// TwinCAT 3 PLC project Area2
// ProgramVersion: 3.1.4023.0
// libraries:
//   Tc2_DataExchange, * (Beckhoff Automation GmbH)
//   Tc2_MC2, * (Beckhoff Automation GmbH)
//   Tc2_Standard, * (Beckhoff Automation GmbH)
//   Tc2_System, * (Beckhoff Automation GmbH)
//   Tc2_TcpIp, * (Beckhoff Automation GmbH)
//   Tc2_Utilities, * (Beckhoff Automation GmbH)
//   Tc3_BA_Common, * (Beckhoff Automation GmbH)
//   Tc3_Database, * (Beckhoff Automation GmbH)
//   Tc3_JsonXml, * (Beckhoff Automation GmbH)
//   Tc3_Module, * (Beckhoff Automation GmbH)
//   Tc3_PackML_V2, * (Beckhoff Automation GmbH)
// project tree:
//   COMMs_ADS/ AdsClient.TcPOU (not stored), AdsHandle.TcPOU
//   COMMs_ADS/PROTOTYPE/ AdsClient_1.TcPOU (not stored), AdsHandle_1.TcPOU (not stored)
//   COMMs_TCP/ TcpServer1Vision.TcPOU
//   COMMs_TCP/Types/ DUT.TcDUT, TcpData.TcDUT (not stored), TcpDataQueue.TcPOU
//   DUTs/Enums/ E_PMLCustomUnitMode.TcDUT (not stored), InsertionDirection.TcDUT, SectionEnum.TcDUT (not stored), SectionTask.TcDUT (not stored), ConveyorMode.TcDUT (not stored), Cover.TcDUT (not stored), EventsEnum.TcTLEO (not stored), MaterialEnums.TcDUT, MaterialType.TcDUT (not stored), Surface.TcDUT (not stored)
//   DUTs/Enums/Materials/ Cardboard.TcDUT, Chipboard.TcDUT, CornerGuard.TcDUT (not stored), WoodBunk.TcDUT (not stored)
//   DUTs/Enums/Robot Tasks/ TaskA22.TcDUT (not stored), TaskA26.TcDUT, TaskA21.TcDUT
//   DUTs/Hardware/ A21ToolStorage.TcDUT (not stored), ConveyorLSC.TcPOU (not stored), ConveyorSC.TcPOU (not stored), FoldingMachine.TcDUT (not stored), PMLStackLight.TcPOU (not stored), Conveyor.TcPOU (not stored)
//   DUTs/Hardware/Big Machines/ StrapMachine.TcPOU (not stored), WrapMachine.TcPOU
//   DUTs/Hardware/Insertion Package/Drives/ AirPiston.TcPOU (not stored), ClearLinkMC.TcPOU, ServoNC.TcPOU (not stored), SimplePiston.TcPOU (not stored)
//   DUTs/Hardware/Insertion Package/ Homing.TcDUT (not stored), Insertion.TcPOU, SuctionPad.TcDUT (not stored)
//   DUTs/Hardware/Insertion Package/Prototypes/ FBA_Drive.TcPOU (not stored), FBA_TrifectaDrive.TcPOU (not stored), I_ContinuousDrive.TcIO (not stored), I_Drive.TcIO (not stored), I_EncodedDrive.TcIO, I_PositionalDrive.TcIO (not stored)
//   DUTs/Hardware/Material Holders/ MaterialHolder.TcPOU (not stored), MaterialSlot.TcDUT (not stored), SkidMagazine.TcPOU (not stored), StagingTable.TcPOU
//   DUTs/Hardware/Robots/ KukaRobot.TcPOU, RobotA21.TcPOU (not stored), RobotA26.TcPOU, RobotA22.TcPOU (not stored)
//   DUTs/ Watchdog.TcPOU, ONE_BIT.TcDUT (not stored), VisionFrame.TcDUT (not stored), VisionSuite.TcDUT (not stored)
//   COMMs_ADS/Types/ AdsSocket.TcPOU (not stored), AdsDataQueue.TcPOU, AdsData.TcDUT
//   DUTs/Bundle/ Bundle.TcDUT, CardboardMaterial.TcDUT, Interval.TcDUT, Material.TcDUT, PositionMaterials.TcDUT (not stored)
//   DUTs/Containers/ DynamicQueue.TcPOU, PtrQueue.TcPOU, IntQueue.TcPOU, Queue.TcPOU, StringQueue.TcPOU
//   EventLogging/ EventLogger.TcIO, SqlDatabaseAccessor.TcPOU (not stored)
//   / GlobalTextList.TcGTLO (not stored), PlcTask.TcTTO (not stored)
//   GVLs/ GVL.TcGVL, CONSTS.TcGVL
//   HARDWARE_DISTRUBUTION/ ConveyorControlModule.TcPOU, ConveyorSyncUnit.TcPOU, A21.TcPOU, A22.TcPOU, A23.TcPOU, A24.TcPOU, A25.TcPOU, A26.TcPOU
//   POUs/Helper Functions/Document/ CreateJsonDocumentManual.TcPOU (not stored), CreateJsonDocumentAuto.TcPOU (not stored), FrameIsValid.TcPOU (not stored), VisionJsonParser.TcPOU (not stored)
//   POUs/Helper Functions/General/ BufferIsEmpty.TcPOU, BundleIsValid.TcPOU (not stored), InRange.TcPOU (not stored), PositionIsValid.TcPOU (not stored), TimestructToString.TcPOU
//   POUs/Helper Functions/Hardware Modules/ InsertionQuality.TcPOU (not stored), SetSuctions.TcPOU, SetSuctionsPtr.TcPOU, SetupHardware.TcPOU, SuctionQuality.TcPOU (not stored), SuctionQualityPtr.TcPOU
//   POUs/Helper Functions/Material Functions/ GetPairMasterLength.TcPOU, GetMaterialLength.TcPOU, MatchesMaterialType.TcPOU (not stored)
//   POUs/Helper Functions/Other/ ForceSetLifterConveyors.TcPOU (not stored), SizeCheck.TcPOU (not stored)
//   POUs/Helper Functions/Utility/ AddToStringArray.TcPOU (not stored), DataIsEmpty.TcPOU (not stored), CleanStringsArray.TcPOU (not stored), IntegerBitAccess.TcPOU (not stored), IntegerToBoolArray.TcPOU (not stored), JoinStrings.TcPOU (not stored), WithinTolerance.TcPOU (not stored)
//   POUs/ MAIN.TcPOU
//   Sections/A21a - Chipboard/AOIs/ AOI_LoadChipboard.TcPOU
//   Sections/A21a - Chipboard/ ChipboardEx.TcPOU
//   Sections/A21b - Wood Bunk/AOIs/ AOI_LoadWoodBunk.TcPOU, AOI_StageWoodBunk.TcPOU (not stored), AOI_StagingTemplate.TcPOU
//   Sections/A21b - Wood Bunk/ WoodBunkEx.TcPOU
//   Sections/A22 - Cardboard/AOIs/ AOI_LoadCornerCardboard.TcPOU, AOI_LoadCornerGuard.TcPOU, AOI_LoadFlatCardboard.TcPOU
//   Sections/A22 - Cardboard/ CardboardEx.TcPOU
//   Sections/A26 - Spacer Recollection/ SpacerRecollectionUnit.TcPOU
//   Sections/Abstract/ SectionEx.TcPOU
// real-time tasks:
//   TASK PlcTask: cycle T#10ms, priority 20, ADS port 350

// ---- COMMs_TCP/Types/DUT.TcDUT
TYPE DUT :
UNION
END_UNION
END_TYPE

// ---- DUTs/Enums/InsertionDirection.TcDUT
{attribute 'qualified_only'}
{attribute 'strict'}
TYPE InsertionDirection :
(
	IN,
	OUT,
	
	size
);
END_TYPE

// ---- DUTs/Enums/Materials/Cardboard.TcDUT
{attribute 'qualified_only'}
{attribute 'to_string'}
TYPE Cardboard :
(
	CAR20S := 1,
	CAR20M,
	CAR20L,
	
	CAR28S,
	CAR28M,
	CAR28L,
	
	size
);
END_TYPE

// ---- DUTs/Enums/Materials/Chipboard.TcDUT
{attribute 'qualified_only'}
{attribute 'to_string'}
TYPE Chipboard :
(
	CIP18 := 1,
	CIP54,
	
	size
);
END_TYPE

// ---- DUTs/Enums/Robot Tasks/TaskA26.TcDUT
{attribute 'qualified_only'}
{attribute 'to_string'}
//{attribute 'strict'}
TYPE TaskA26 :
(
	IDLE,
	PICK_SPACER,
	
	size
);
END_TYPE

// ---- DUTs/Enums/Robot Tasks/TaskA21.TcDUT
{attribute 'qualified_only'}
//{attribute 'strict'}
{attribute 'to_string'}
TYPE TaskA21 :
(
	IDLE,
	STAGE_BUNK,
	REMOVE_BUNK_FROM_STAGE,
	
	LOAD_BUNK_TOP := 4,
	LOAD_BUNK_SIDE,
	LOAD_BUNK_BOTTOM,
	REMOVE_BUNK_TOP,
	REMOVE_BUNK_SIDE,
	REMOVE_BUNK_BOTTOM,
	
	//GET_CHIPBOARD_FROM_SKID := 11,
	//OFFLOAD_CHIPBOARD,
	PLACE_CHIPBOARD_TOP := 13,
	PLACE_CHIPBOARD_BOTTOM,
	REMOVE_CHIPBOARD_TOP,
	REMOVE_CHIPBOARD_BOTTOM,
	
	FIX_CHIPBOARD_ORIENTATION := 19,
	
	//testing only
	MOVE_HOME := 21,
	MOVE_POSITION1,
	MOVE_POSITION2,
	MOVE_UP,
	MOVE_DOWN,
	
	DIRECT_BUNK_TOP := 27,
	DIRECT_BUNK_SIDE,
	DIRECT_BUNK_BOTTOM,
	
	INSPECT_BUNK := 31,
	INSPECT_CHIPBOARD,
	
	TOOL_CHANGE_BUNK := 34,
	TOOL_CHANGE_CHIPBOARD,
	
	size
);
END_TYPE

// ---- COMMs_ADS/Types/AdsData.TcDUT
{attribute 'enable_dynamic_creation'}
TYPE AdsData :
STRUCT	
	description : EventsEnum; //purpose
	
	timestamp : TIMESTRUCT; //relevant timestamp (ex: arrival time)
	
	binaryData : ARRAY[0..100000] OF BYTE; //contents
END_STRUCT
END_TYPE

// ---- DUTs/Bundle/Bundle.TcDUT
{attribute 'enable_dynamic_creation'}
TYPE Bundle :
STRUCT
	id : STRING;
	weight : REAL;
	
	length : INT;
	width : INT;
	height : INT;
	
	pieces : INT;
	layers : INT;
	piecesPerLayer : INT;
	
	extrusionWeight : INT;
	extrusionHeight : INT;
	extrusionWidth : INT;
	
	//if a process is true, send it to the correct area and turn it false when complete
	reqProcesses : ARRAY[0..3] OF BOOL;
	
	manRE, autoRE : BOOL; //repacking - coming soon
	manSS, autoSS : BOOL; //packaging
	
	currStep : USINT; //for runtime use only
	
	paperFront : BOOL;
	paperBack : BOOL;
	cardboardFront : BOOL;
	cardboardBack : BOOL;
	
	paperTop : ARRAY[0..Consts.maxPairs] OF Interval;
	paperLeft : ARRAY[0..Consts.maxPairs] OF Interval;
	paperRight : ARRAY[0..Consts.maxPairs] OF Interval;
	paperBottom : ARRAY[0..Consts.maxPairs] OF Interval;
		
	cardboard : ARRAY[0..Consts.maxPairs] OF PositionMaterials;
	cardboardFolds : ARRAY[Surface.TOP_LEFT..Surface.BOTTOM_RIGHT] OF ARRAY[0..Consts.maxPairs] OF INT;
	
	topLeftFolds : ARRAY[0..Consts.maxPairs] OF INT;
	topRightFolds : ARRAY[0..Consts.maxPairs] OF INT;
	bottomLeftFolds : ARRAY[0..Consts.maxPairs] OF INT;
	bottomRightFolds : ARRAY[0..Consts.maxPairs] OF INT;
	
	cornerGuard : ARRAY[0..Consts.maxPairs] OF PositionMaterials;
	
	chipboard : ARRAY[0..Consts.maxPairs] OF PositionMaterials;
	woodBunk : ARRAY[0..Consts.maxPairs] OF PositionMaterials;
	
	cardboard_over_cornerGuard : BOOL;
	
	//for production log database
	timeStart : TIMESTRUCT;
	timeDone : TIMESTRUCT;
END_STRUCT
END_TYPE

// ---- DUTs/Bundle/CardboardMaterial.TcDUT
TYPE CardboardMaterial :
STRUCT
	foldType : (FLAT, CORNER, COVER);
	foldPos1 : REAL;
	foldPos2 : REAL;
END_STRUCT
END_TYPE

// ---- DUTs/Bundle/Interval.TcDUT
TYPE Interval :
STRUCT
	startPos : INT;
	endPos : INT;
END_STRUCT
END_TYPE

// ---- DUTs/Bundle/Material.TcDUT
TYPE Material :
STRUCT
	code : STRING;
	width : REAL;
	length : REAL;
END_STRUCT
END_TYPE
(*
use this struct to keep track of where materials are
materials enter the system when pulled from their magazine/skid and exit the system when placed on the bundle or otherwise lost
*)

// ---- DUTs/Enums/MaterialEnums.TcDUT
{attribute 'qualified_only'}
{attribute 'strict'}
{attribute 'to_string'}
TYPE MaterialEnums :
(
	//CARDBOARD - 6 x 3
	CAR20S, CAR20M, CAR20L, CAR28S, CAR28M, CAR28L, //base (flat)
	CAR20SF, CAR20MF, CAR20LF, CAR28SF, CAR28MF, CAR28LF, //single folded (L shape) - F
	CAR20SD, CAR20MD, CAR20LD, CAR28SD, CAR28MD, CAR28LD, //double folded (C shape) - D
	
	//CHIPBOARD - 2
	CIP18, CIP54,
	
	//CORNER BOARD - 2
	COR48, COR96,
	
	//PAPER - 1
	PAP28,
	
	//WOOD BUNK - 21
	WDT20, WDT22, WDT28, //top
	WDB20, WDB22, WDB28, //bottom
	WDS08, WDS10, WDS12, WDS14, WDS20, WDS22, WDS28, //side
	WDS8X8, WDS8X10, WDS12X12, WDS12X14, WDS20X10, WDS20X12, //side combined - X
	WDW20, WDW22, //special top (wide)
	
	size //number of materials
);
END_TYPE

// ---- GVLs/GVL.TcGVL
{attribute 'qualified_only'}
VAR_GLOBAL
	bundleOut : Bundle; //may or may not be used?
	
	iecCriticalSection : FB_IecCriticalSection; //must be used if communication routines are separated into their own core/task
END_VAR

// ---- GVLs/CONSTS.TcGVL
{attribute 'qualified_only'}
VAR_GLOBAL CONSTANT
	maxPairs : USINT := 16;
	initArraySize : USINT := 4;
	maxQueue : INT := 16;
	
	nullPos : REAL := -1;
	
	numMaterials : INT := 32;
	allMaterials : ARRAY[0..numMaterials] OF Material := [
		(code := '', width := 0, length := 0), //null material
		(code := 'PAP28', width := 28, length := -1),
		
		(code := 'CAR20S', width := 20, length := 30),
		(code := 'CAR20M', width := 20, length := 45),
		(code := 'CAR20L', width := 20, length := 60),
		(code := 'CAR28S', width := 28, length := 30),
		(code := 'CAR28M', width := 28, length := 45),
		(code := 'CAR28L', width := 28, length := 60),
		
		(code := 'COR48', width := 1.5, length := 48),
		(code := 'COR96', width := 1.5, length := 96),
		
		(code := 'CIP18', width := 20, length := 18),
		(code := 'CIP54', width := 20, length := 54),
		
		(code := 'WDT20', width := 20, length := 2.5),
		(code := 'WDT22', width := 22, length := 2.5),
		(code := 'WDT28', width := 28, length := 2.5),
		
		(code := 'WDB20', width := 20, length := 2.5),
		(code := 'WDB22', width := 22, length := 2.5),
		(code := 'WDB28', width := 28, length := 2.5),
		
		(code := 'WDS08', width := 8, length := 2.5),
		(code := 'WDS10', width := 10, length := 2.5),
		(code := 'WDS12', width := 12, length := 2.5),
		(code := 'WDS14', width := 14, length := 2.5),
		(code := 'WDS8x8', width := 16, length := 2.5),
		(code := 'WDS8x10', width := 18, length := 2.5),
		(code := 'WDS20', width := 20, length := 2.5),
		(code := 'WDS22', width := 22, length := 2.5),
		(code := 'WDS12x12', width := 24, length := 2.5),
		(code := 'WDS12x14', width := 26, length := 2.5),
		(code := 'WDS28', width := 28, length := 2.5),
		(code := 'WDS20x10', width := 30, length := 2.5),
		(code := 'WDS20x12', width := 32, length := 2.5),
		
		(code := 'WDW20', width := 20, length := 6),
		(code := 'WDW22', width := 22, length := 6)];

	//nullBundle : Bundle;
	
	//conveyorLength : REAL := 0;
	precisionTolerance : REAL := 0.05 * 25.4;
END_VAR
VAR_GLOBAL CONSTANT
	numTotalConveyors : INT := 38;
	
	numCellConveyors : INT := 20;
	
	numReceiverConveyors : INT := 6;
	numOutputConveyors : INT := 12;
END_VAR

// ---- DUTs/Hardware/Insertion Package/Prototypes/I_EncodedDrive.TcIO
INTERFACE I_EncodedDrive EXTENDS I_PositionalDrive, I_ContinuousDrive
//this drive can perform absolute/relative targeting and continuous motion
//only used if a drive with both encoded and continuous behavior is needed

END_INTERFACE

// ---- EventLogging/EventLogger.TcIO
INTERFACE EventLogger

METHOD logEvent : BOOL
VAR_INPUT
END_VAR
END_METHOD

METHOD queueEvent : BOOL
VAR_INPUT
	event : INT;
END_VAR
END_METHOD

END_INTERFACE

// ---- COMMs_ADS/AdsHandle.TcPOU
FUNCTION_BLOCK AdsHandle
VAR_INPUT
	ServerNetId			: STRING; 	(* Server AmsNetId *)
	ServerPort 			: UDINT;	(* Server port number *)
	
	remoteAccessPrefix	: STRING;
END_VAR
VAR_OUTPUT
	bBusy				: BOOL;
	err					: BOOL;
	errid				: UDINT;
	
	receiveBuffer		: ARRAY[0..100000] OF BYTE; //TCP style data buffer
	receiveStruct		: AdsData;
END_VAR
VAR	
	socket 				: AdsSocket; //only this needs initialization
	
	sendQueue			: AdsDataQueue;
	sendBufferQueue 	: DynamicQueue; //anything going into this needs to be a TcpStruct
	
	sendBuffer 			: ARRAY[0..50000] OF BYTE; //temp byte buffer to send if neccessary
	sendStruct			: AdsData;
	
	//setupStep 			: (CLOSE_CONNECTIONS, CREATE_LISTENER, ACCEPT_CONNECTION, FINISH_SETUP);
	sendDelay : TON;
END_VAR
VAR_STAT CONSTANT
	sendDelayTime : TIME := T#1S;
END_VAR

sendDelay(IN:= , PT:= sendDelayTime, Q=> , ET=> );
sendDelay.IN := TRUE;

IF sendDelay.Q THEN
	
	sendStruct := sendQueue.poll();
	IF NOT DataIsEmpty(arr := ADR(sendStruct), arrSize := SIZEOF(sendStruct)) THEN //if valid data to send	
		write(
			symbol := CONCAT(remoteAccessPrefix, 'receiveStruct'),
			data := ADR(sendStruct),
			dataSize := SIZEOF(sendStruct));
			
		sendDelay.IN := FALSE;
	END_IF
	
END_IF

METHOD clearBuffer : BOOL
VAR
	emptyReceiverStruct : AdsData;
END_VAR
//MEMSET(ADR(receiveBuffer), 0, SIZEOF(receiveBuffer));
receiveStruct := emptyReceiverStruct;
END_METHOD

METHOD close : BOOL
VAR_INPUT
END_VAR
socket.close();
END_METHOD

METHOD getHandlerName : STRING
getHandlerName := socket.remotePrgName;
END_METHOD

METHOD open : BOOL
VAR_INPUT
	localPrgName : STRING;
	localNetId : T_AmsNetId;
	localPort : T_AmsPort;
END_VAR
socket.open(localPrgName, localNetId, localPort);
END_METHOD

METHOD queueData : BOOL
VAR_INPUT
	data : REFERENCE TO AdsData;
END_VAR
//MEMCPY(ADR(temp), data.pValue, data.diSize);
sendQueue.push(data);
END_METHOD

METHOD read : BOOL
VAR_INPUT
	symbol : STRING;
	buffer : PVOID;
	symbolSize : UDINT;
END_VAR
IF NOT socket.readBusy THEN
	read := socket.read(
		symbol:= symbol,
		buffer := buffer,
		symbolSize := symbolSize);
END_IF
END_METHOD

METHOD write : BOOL
VAR_INPUT
	symbol : STRING;
	data : PVOID;
	dataSize : UDINT;
END_VAR
VAR
	timer : TON;
END_VAR
IF NOT socket.writeBusy THEN
	write := socket.write(
		symbol:= symbol,
		data := data,
		dataSize := dataSize);
END_IF
END_METHOD

END_FUNCTION_BLOCK

// ---- COMMs_ADS/Types/AdsDataQueue.TcPOU
{attribute 'call_after_init'}
FUNCTION_BLOCK AdsDataQueue
VAR
	elements : FB_BA_DynamicArray := (uiEntrySize := SIZEOF(POINTER TO AdsData), uiMinExpCount := CONSTS.initArraySize); 
	length : INT := 0;
	
	entrySize : UDINT;
END_VAR
(*
this container stores dynamically generated AdsData Structs
AdsData to be added are passed by reference, then this function block allocates a structure to be stored
AdsData are get() by reference and poll() by value
*)

METHOD clear : BOOL
VAR
	i : INT;
	temp : REFERENCE TO AdsData;
	tempAdr : POINTER TO AdsData;
END_VAR
FOR i:=0 TO length-1 BY 1 DO
	temp := get(index := i, getSize => );
	tempAdr := ADR(temp);
	__DELETE(tempAdr);
END_FOR

elements.Reset();
length := 0;
END_METHOD

METHOD contains : BOOL //check contents, not pointer value
VAR_INPUT
	value : REFERENCE TO AdsData;
END_VAR
VAR_OUTPUT
	atIndex : INT;
END_VAR
VAR
	temp : REFERENCE TO AdsData;
	i : INT;
END_VAR
IF length = 0 THEN
	contains := FALSE;
	RETURN;
END_IF

FOR i:=0 TO length-1 BY 1 DO
	temp := get(index := i, getSize => );
	
	IF 
		SIZEOF(value) = entrySize AND //same size
		MEMCMP(ADR(temp), ADR(value), SIZEOF(entrySize)) = 0 //same data
	THEN
		contains := TRUE;
		atIndex := i;
		RETURN;
	END_IF
	
END_FOR
contains := FALSE;
END_METHOD

METHOD get : REFERENCE TO AdsData
VAR_INPUT
	index : INT;
END_VAR
VAR_OUTPUT
	getSize : UDINT;
END_VAR
IF length = 0 OR index < 0 OR index >= length THEN
	getSize := 0;
ELSE
	elements.GetEntry(diIndex := index, pResultEntry := ADR(get));
	getSize := SIZEOF(get);
END_IF
END_METHOD

METHOD isEmpty : BOOL
VAR_INPUT
END_VAR
isEmpty := length = 0;
END_METHOD

METHOD poll : AdsData
VAR_OUTPUT
	getSize : UDINT;
END_VAR
IF length > 0 THEN
	poll := get(index := 0, getSize => getSize);
	elements.RemoveEntry(diIndex := 0);
	
	length := length - 1;
END_IF
END_METHOD

METHOD push : BOOL
VAR_INPUT
	value : REFERENCE TO AdsData;
END_VAR
VAR
	temp : POINTER TO AdsData;
END_VAR
temp := __NEW(AdsData);
temp^ := value;

elements.AddEntryPtr(pEntry := temp);

length := length + 1;
END_METHOD

METHOD set : BOOL
VAR_INPUT
	i : INT;
	value : REFERENCE TO AdsData;
END_VAR
VAR
	temp : REFERENCE TO AdsData;
END_VAR
IF length = 0 THEN
	RETURN;
END_IF

IF i >= 0 AND i < length THEN
	temp REF= get(i);
	temp := value;
	
	set := TRUE;
END_IF
END_METHOD

{attribute 'call_after_init'}
METHOD setup : BOOL
VAR_INPUT
END_VAR
entrySize := SIZEOF(AdsData);
END_METHOD

METHOD size : INT
size := length;
END_METHOD

END_FUNCTION_BLOCK

// ---- DUTs/Containers/DynamicQueue.TcPOU
FUNCTION_BLOCK DynamicQueue
VAR
	elements : FB_BA_DynamicArray := (uiEntrySize := SIZEOF(POINTER TO BYTE), uiMinExpCount := CONSTS.initArraySize); 
	elementSizes : FB_BA_DynamicArray := (uiEntrySize := SIZEOF(LINT), uiMinExpCount := CONSTS.initArraySize);
	length : INT := 0;
END_VAR
(*
this dynamic array stores pointers to dynamically generated objects
elements to be added are passed by value, then this function block allocates bytes
*)

METHOD clear : BOOL
VAR
	i : INT;
	temp : POINTER TO BYTE;
END_VAR
FOR i:=0 TO length-1 BY 1 DO
	temp := get(index := i);
	__DELETE(temp);
END_FOR


elements.Reset();
elementSizes.Reset();
length := 0;
END_METHOD

METHOD contains : BOOL
VAR_INPUT
	value : ANY;
END_VAR
VAR_OUTPUT
	atIndex : INT;
END_VAR
VAR
	temp : POINTER TO BYTE;
	tempSize : LINT;
	i : INT;
END_VAR
IF length = 0 THEN
	contains := FALSE;
	RETURN;
END_IF

FOR i:=0 TO length-1 BY 1 DO
	temp := get(index := i, getSize => tempSize);
	
	IF 
		tempSize = value.diSize AND //same size
		MEMCMP(get(i), value.pValue, TO_UDINT(value.diSize)) = 0 //same data
	THEN
		contains := TRUE;
		atIndex := i;
		RETURN;
	END_IF
	
END_FOR
contains := FALSE;
END_METHOD

METHOD get : POINTER TO BYTE
VAR_INPUT
	index : INT;
END_VAR
VAR_OUTPUT
	getSize : LINT;
END_VAR
IF length = 0 OR index < 0 OR index >= length THEN
	get := 0;
	getSize := 0;
ELSE
	elements.GetEntry(diIndex := index, pResultEntry := ADR(get));
	elementSizes.GetEntry(diIndex := index, pResultEntry := ADR(getSize));
END_IF
END_METHOD

METHOD isEmpty : BOOL
VAR_INPUT
END_VAR
isEmpty := length = 0;
END_METHOD

METHOD poll : POINTER TO BYTE
VAR_OUTPUT
	getSize : LINT;
END_VAR
poll := get(index := 0, getSize => getSize);

IF length > 0 THEN
	elements.RemoveEntry(diIndex := 0);
	elementSizes.RemoveEntry(diIndex := 0);
	
	length := length - 1;
END_IF
END_METHOD

METHOD push : BOOL
VAR_INPUT
	value : ANY;
END_VAR
VAR
	temp : POINTER TO BYTE;
END_VAR
temp := __NEW(BYTE, TO_UDINT(value.diSize));
MEMCPY(temp, value.pValue, TO_UDINT(value.diSize));

elements.AddEntryPtr(pEntry := temp);
elementSizes.AddEntry(pEntry := ADR(value.diSize));

length := length + 1;
END_METHOD

METHOD set : BOOL
VAR_INPUT
	i : INT;
	value : ANY;
END_VAR
VAR
	temp : POINTER TO BYTE;
	tempSize : UDINT;
END_VAR
IF length = 0 THEN
	RETURN;
END_IF

IF i >= 0 AND i < length THEN
	temp := get(i);
	__DELETE(temp);
	
	tempSize := TO_UDINT(value.diSize);
	temp := __NEW(BYTE, tempSize);
	MEMCPY(temp, value.pValue, tempSize);

	elements.SetEntryPtr(i, ADR(temp));
	elementSizes.SetEntry(i, ADR(tempSize)); 
	set := TRUE;
END_IF
END_METHOD

METHOD size : INT
size := length;
END_METHOD

END_FUNCTION_BLOCK

// ---- COMMs_TCP/TcpServer1Vision.TcPOU
PROGRAM TcpServer1Vision
VAR_INPUT
	ServerNetId			: STRING; 	(* Server AmsNetId *)
	ServerAdr 			: STRING;	(* Server IP address *)
	ServerPort 			: UDINT;	(* Server port number *)
END_VAR
VAR_OUTPUT
	busy				: BOOL;
	error				: BOOL;
	errorId				: UDINT;
	bytesReceived		: UDINT;
	
	receiveStruct		: TcpData;	(* Data received *)
	connected 			: BOOL;
END_VAR
VAR
	fbSocketCloseAll 	: FB_SocketCloseAll;
	fbSocketClose 		: FB_SocketClose;
	
	fbSocketListen		: FB_SocketListen;
	fbSocketAccept		: FB_SocketAccept;
	fbSocketReceive		: FB_SocketReceive;
	fbSocketSend 		: FB_SocketSend;
	
	listenerSocket		: T_HSOCKET;
	dataSocket			: T_HSOCKET;
	
	sendQueue 			: TcpDataQueue;
	sendBuffer 			: ARRAY[0..99] OF BYTE;
	
	sendHeartbeats		: BOOL;
	autoDisconnect		: BOOL;
	
	setupStep 			: (CLOSE_CONNECTIONS, CREATE_LISTENER, ACCEPT_CONNECTION, FINISH_SETUP);
	
	setupTimer : TON;
	connectionTimer	: TON;
	heartbeatTimer : TON;
END_VAR
VAR CONSTANT
	connectionTimeout	: TIME := T#30S; //time before connection is closed
	heartbeatInterval	: TIME := T#20S; //heartbeat intervals
	
	incomingHeartbeat	: STRING := 'HEARTBEAT_CLIENT_TO_SERVER';
	outgoingHeartbeat	: STRING := 'HEARTBEAT_SERVER_TO_CLIENT';
END_VAR

blocks();

connected := setup();
IF NOT connected THEN
	RETURN;
END_IF

receive(); //receive in real time

IF autoDisconnect THEN
	autoDisconnectSeq();
ELSE
	connectionTimer.IN := FALSE;
END_IF

IF sendHeartbeats THEN
	sendHeartbeatSeq();
ELSE
	heartbeatTimer.IN := FALSE;
END_IF

send();

METHOD PRIVATE autoDisconnectSeq : BOOL
connectionTimer(IN := , PT := connectionTimeout, Q => , ET => );
connectionTimer.IN := TRUE;

IF connectionTimer.Q THEN
	connectionTimer.IN := FALSE;
	
	closeSocket(dataSocket);
	//closeSocket(listenerSocket);
	
	setupStep := CLOSE_CONNECTIONS;
	RETURN;
END_IF
END_METHOD

METHOD PRIVATE blocks : BOOL
fbSocketClose(
	sSrvNetId:= ServerNetId, 
	hSocket:= dataSocket, 
	bExecute:= , 
	tTimeout:= , 
	bBusy=> busy, 
	bError=> error, 
	nErrId=> errorId);
	
fbSocketCloseAll(
	sSrvNetId:= ServerNetId, 
	bExecute:= , 
	tTimeout:= , 
	bBusy=> , 
	bError=> , 
	nErrId=> );
	
IF fbSocketClose.bExecute OR fbSocketCloseAll.bExecute THEN
	fbSocketClose.bExecute := FALSE;
	fbSocketCloseAll.bExecute := FALSE;
END_IF
	
fbSocketListen(
	sSrvNetId:= ServerNetId, 
	sLocalHost:= ServerAdr, 
	nLocalPort:= ServerPort, 
	bExecute:= , 
	tTimeout:= , 
	bBusy=> busy, 
	bError=> error, 
	nErrId=> errorId, 
	hListener=> listenerSocket);

fbSocketAccept(
	sSrvNetId:= ServerNetId, 
	hListener:= listenerSocket, 
	bExecute:= , 
	tTimeout:= , 
	bAccepted=> , 
	bBusy=> busy, 
	bError=> error, 
	nErrId=> errorId, 
	hSocket=> dataSocket);
	
fbSocketReceive(
	sSrvNetId:= ServerNetId, 
	hSocket:= dataSocket, 
	cbLen:= SIZEOF(receiveStruct), 
	pDest:= ADR(receiveStruct), 
	bExecute:= , 
	tTimeout:= , 
	bBusy=> busy, 
	bError=> error, 
	nErrId=> errorId, 
	nRecBytes=> bytesReceived);
	
fbSocketSend(
	sSrvNetId:= ServerNetId, 
	hSocket:= dataSocket, 
	cbLen:= SIZEOF(sendBuffer), 
	pSrc:= ADR(sendBuffer), 
	bExecute:= , 
	tTimeout:= ,
	bBusy=> busy, 
	bError=> error, 
	nErrId=> errorId);
END_METHOD

METHOD PRIVATE clearBuffer : BOOL
MEMSET(ADR(receiveStruct), 0, SIZEOF(receiveStruct));
END_METHOD

METHOD PRIVATE closeSocket : BOOL
VAR_INPUT
	socket : REFERENCE TO T_HSOCKET;
END_VAR
fbSocketClose.bExecute := TRUE;
fbSocketClose.hSocket := socket;
END_METHOD

METHOD fetch : BOOL
VAR_IN_OUT
	receiverStruct : TcpData;
END_VAR
VAR
	emptyData : TcpData;
END_VAR
fetch := MEMCMP(ADR(receiveStruct), ADR(emptyData), SIZEOF(TcpData)) <> 0; //returns false if no data

receiverStruct := receiveStruct;
receiveStruct := emptyData;
END_METHOD

METHOD queue : BOOL
VAR_INPUT
	data : REFERENCE TO TcpData;
END_VAR
sendQueue.push(data);
END_METHOD

METHOD PRIVATE receive : BOOL
VAR
	heartbeatCheck : STRING;
END_VAR
fbSocketReceive.bExecute := NOT fbSocketReceive.bExecute;
	
MEMCPY(ADR(heartbeatCheck), ADR(receiveStruct), SIZEOF(heartbeatCheck));
IF heartbeatCheck = incomingHeartbeat THEN
	connectionTimer.IN := FALSE;
END_IF
END_METHOD

METHOD PRIVATE send : BOOL
VAR
	polledData : TcpData;
END_VAR
IF NOT fbSocketSend.bBusy THEN
	polledData := sendQueue.poll();
	MEMCPY(ADR(sendBuffer), ADR(polledData), MIN(SIZEOF(polledData), SIZEOF(sendBuffer)));
END_IF

IF NOT BufferIsEmpty(sendBuffer) THEN
	fbSocketSend.bExecute := NOT fbSocketSend.bExecute;
	
ELSE
	fbSocketSend.bExecute := FALSE;
	
END_IF
END_METHOD

METHOD PRIVATE sendHeartbeatSeq : BOOL
VAR
	temp : TcpData;
END_VAR
heartbeatTimer(IN := , PT := heartbeatInterval, Q =>, ET =>);
heartbeatTimer.IN := TRUE;

IF heartbeatTimer.Q THEN
	MEMCPY(ADR(temp), ADR(outgoingHeartbeat), SIZEOF(outgoingHeartbeat));
	queue(temp);
	
	heartbeatTimer.IN := FALSE;
END_IF
END_METHOD

METHOD PRIVATE setup : BOOL
CASE setupStep OF
	CLOSE_CONNECTIONS:
		fbSocketCloseAll( bExecute:= TRUE );
		fbSocketCloseAll( bExecute:= FALSE );
		setupStep := CREATE_LISTENER;
		
	CREATE_LISTENER:
		fbSocketListen.bExecute := TRUE;
		setupStep := ACCEPT_CONNECTION;
		
	ACCEPT_CONNECTION:
		fbSocketListen.bExecute := FALSE;
		IF fbSocketListen.bError THEN
			setupStep := CLOSE_CONNECTIONS;
			RETURN;
			
		ELSIF NOT fbSocketListen.bBusy AND NOT fbSocketListen.bError THEN
			fbSocketAccept.bExecute := FALSE;
			setupTimer(IN:= , PT:= T#500MS, Q=> , ET=> );
			setupTimer.IN := TRUE;
			IF setupTimer.Q THEN
				fbSocketAccept.bExecute := TRUE;
				setupTimer.IN := FALSE;
			END_IF
		
			IF fbSocketAccept.bAccepted THEN
				setupTimer.IN := FALSE;
				setupStep := FINISH_SETUP;
			END_IF
		END_IF
		
		
	FINISH_SETUP:
		setup := TRUE;
		//fbSocketClose(bExecute := TRUE);
END_CASE
END_METHOD

END_PROGRAM

// ---- COMMs_TCP/Types/TcpDataQueue.TcPOU
{attribute 'call_after_init'}
FUNCTION_BLOCK TcpDataQueue
VAR
	elements : FB_BA_DynamicArray := (uiEntrySize := SIZEOF(POINTER TO TcpData), uiMinExpCount := CONSTS.initArraySize); 
	length : INT := 0;
	
	entrySize : UDINT;
END_VAR
(*
this container stores dynamically generated AdsData Structs
AdsData to be added are passed by reference, then this function block allocates a structure to be stored
AdsData are get() by reference and poll() by value
*)

METHOD clear : BOOL
VAR
	i : INT;
	temp : REFERENCE TO TcpData;
	tempAdr : POINTER TO TcpData;
END_VAR
FOR i:=0 TO length-1 BY 1 DO
	temp := get(index := i, getSize => );
	tempAdr := ADR(temp);
	__DELETE(tempAdr);
END_FOR

elements.Reset();
length := 0;
END_METHOD

METHOD contains : BOOL //check contents, not pointer value
VAR_INPUT
	value : REFERENCE TO TcpData;
END_VAR
VAR_OUTPUT
	atIndex : INT;
END_VAR
VAR
	temp : REFERENCE TO TcpData;
	i : INT;
END_VAR
IF length = 0 THEN
	contains := FALSE;
	RETURN;
END_IF

FOR i:=0 TO length-1 BY 1 DO
	temp := get(index := i, getSize => );
	
	IF 
		SIZEOF(value) = entrySize AND //same size
		MEMCMP(ADR(temp), ADR(value), SIZEOF(entrySize)) = 0 //same data
	THEN
		contains := TRUE;
		atIndex := i;
		RETURN;
	END_IF
	
END_FOR
contains := FALSE;
END_METHOD

METHOD get : REFERENCE TO TcpData
VAR_INPUT
	index : INT;
END_VAR
VAR_OUTPUT
	getSize : UDINT;
END_VAR
IF length = 0 OR index < 0 OR index >= length THEN
	getSize := 0;
ELSE
	elements.GetEntry(diIndex := index, pResultEntry := ADR(get));
	getSize := SIZEOF(get);
END_IF
END_METHOD

METHOD isEmpty : BOOL
VAR_INPUT
END_VAR
isEmpty := length = 0;
END_METHOD

METHOD poll : TcpData
VAR_OUTPUT
	getSize : UDINT;
END_VAR
IF length > 0 THEN
	poll := get(index := 0, getSize => getSize);
	elements.RemoveEntry(diIndex := 0);
	
	length := length - 1;
END_IF
END_METHOD

METHOD push : BOOL
VAR_INPUT
	value : REFERENCE TO TcpData;
END_VAR
VAR
	temp : POINTER TO TcpData;
END_VAR
temp := __NEW(TcpData);
temp^ := value;

elements.AddEntryPtr(pEntry := temp);

length := length + 1;
END_METHOD

METHOD set : BOOL
VAR_INPUT
	i : INT;
	value : REFERENCE TO TcpData;
END_VAR
VAR
	temp : REFERENCE TO TcpData;
END_VAR
IF length = 0 THEN
	RETURN;
END_IF

IF i >= 0 AND i < length THEN
	temp REF= get(i);
	temp := value;
	
	set := TRUE;
END_IF
END_METHOD

{attribute 'call_after_init'}
METHOD setup : BOOL
VAR_INPUT
END_VAR
entrySize := SIZEOF(TcpData);
END_METHOD

METHOD size : INT
size := length;
END_METHOD

END_FUNCTION_BLOCK

// ---- DUTs/Containers/Queue.TcPOU
FUNCTION_BLOCK ABSTRACT Queue
VAR
	entrySize : ULINT; //no functionaility, only to force input a type for readability
	length : USINT := 0;
END_VAR

END_FUNCTION_BLOCK

// ---- POUs/Helper Functions/General/BufferIsEmpty.TcPOU
FUNCTION BufferIsEmpty : BOOL
VAR_IN_OUT
	bufferArr : ARRAY[*] OF BYTE;
END_VAR
VAR
	i : DINT;
END_VAR

FOR i:=LOWER_BOUND(bufferArr, 1) TO UPPER_BOUND(bufferArr, 1) BY 1 DO
	IF bufferArr[i] <> 0 THEN
		BufferIsEmpty := FALSE;
		RETURN;
	END_IF
END_FOR
BufferIsEmpty := TRUE;

END_FUNCTION

// ---- DUTs/Hardware/Big Machines/WrapMachine.TcPOU
FUNCTION_BLOCK WrapMachine
VAR_INPUT
	bEnable : BOOL;
	extSafety : BOOL;
END_VAR
VAR_OUTPUT
	error AT %I* : BOOL;
	ready AT %I* : BOOL;
	busy AT %I* : BOOL;
	done (*AT %I**) : BOOL;
	home AT %I* : BOOL;
	
	rotations AT %Q* : INT;
	execute AT %Q* : BOOL;
	enable AT %Q* : BOOL;
	reset AT %Q* : BOOL;
	
	timeout : BOOL;
	
	trayOccupied AT %I* : BOOL;
	overheadMaterial : STRING;
END_VAR
VAR
	holdPost : TON;
	delay : TON;
	
	start : BOOL;
	step : (SETUP, RUN, WAIT);
END_VAR
VAR_STAT CONSTANT
	pulseTime : TIME := T#100MS;
	holdTime : TIME := T#500MS;
	maxDelay : TIME := T#30S;
END_VAR

holdPost(IN:= , PT:= holdTime, Q=> , ET=> );
delay(IN:= step > 0, PT:= maxDelay, Q=> , ET=> );

IF delay.Q THEN
	delay.IN := FALSE;
	timeout := TRUE;
	busy := FALSE;
	step := SETUP;
END_IF

CASE step OF
	SETUP:
		busy := FALSE;
		IF error THEN
			reset := NOT reset;
			enable := FALSE;//NOT enable;
			
		ELSE
			reset := FALSE;
			enable := TRUE;
			
			IF start THEN
				start := FALSE;
				step := RUN;
			END_IF
			
		END_IF
	
	RUN:
		execute := TRUE;
		IF execute AND NOT home THEN
			execute := FALSE;
			step := WAIT;
		END_IF
		
	WAIT:
		IF home THEN
			holdPost.IN := TRUE;
			enable := FALSE;
			execute := FALSE;
		END_IF
		
		IF holdPost.Q THEN
			holdPost.IN := FALSE;
			done := TRUE;
			step := 0;
		END_IF
		
END_CASE

METHOD clear : BOOL
VAR_INPUT
END_VAR
(*
reset should be continuously called until machine returns evidence that it is ready again
machine is expected to not respond to reset signals if it is already in an idle state
*)
enable := FALSE;
execute := FALSE;

IF error THEN
	reset := NOT reset;
	clear := NOT error;

ELSE
	reset := FALSE;
	clear := TRUE;
	
END_IF
END_METHOD

{attribute 'monitoring' := 'call'}
PROPERTY Overhead : STRING
GET
Overhead := overheadMaterial;
END_GET
SET
overheadMaterial := Overhead;
END_SET
END_PROPERTY

METHOD wrap : BOOL
VAR_INPUT
	reqRotations : INT;
END_VAR
IF ready AND NOT busy AND NOT error THEN
	rotations := reqRotations;
	busy := TRUE;
	start := TRUE;
	wrap := TRUE;
END_IF
END_METHOD

END_FUNCTION_BLOCK

// ---- DUTs/Hardware/Insertion Package/Drives/ClearLinkMC.TcPOU
FUNCTION_BLOCK ClearLinkMC EXTENDS FBA_TrifectaDrive IMPLEMENTS I_EncodedDrive
VAR_OUTPUT
	pulse AT %Q* : INT;
	brakeRelease AT %Q* : BOOL := TRUE;
	enable : BOOL;
	A : BOOL;
	B : BOOL;
	clear : BOOL;
END_VAR
VAR	
	hlfb AT %I* : REAL := -9999; //high level feedback, if -9999 then servo is idle
	
	outputRegister AT %Q* : INT;
	pulseRequest : INT;
	
	homingDelay : TON;
	resetPulse : TP;
	
	mode : (HOLD, TARGET, CONTINUOUS, RESET_ERR);
	calculation : (IDLE, DOWN, UP, CALCULATE, DONE);
	maxPosition : LREAL;
	
	position, targetPos : LREAL;
	
	pulsePosition : INT;
	pulseCounter : INT;
	rotationsPerPulse : INT; //revolutions per pulse
	displacementPerPulse : LREAL; //displacement per pulse
END_VAR
VAR_STAT CONSTANT
	resetWidth : TIME := T#500MS;
	delayWidth : TIME := T#500MS;
END_VAR
VAR //constructor
	homingDirectionOut : BOOL; 			//homing direction - see <A>
	minPosition : LREAL;
	displacementPerRotation : LREAL; 	//displacement per revolution	
	unitsPerPulse : INT := 800; 		//800 Teknic units per rotation - default setting is 800 units (1 rotation) per pulse
END_VAR

//M-connector output register
outputRegister.0 := enable AND bEnable; 	//enable
outputRegister.1 := A; 						//direction bit - T = outwards, F = inwards
outputRegister.2 := B; 						//homing bit - after startup, set to TRUE to begin homing, then set to FALSE to finish homing
outputRegister.3 := clear; 					//reset bit

rotationsPerPulse := unitsPerPulse/800; //Teknic constant - 800 units per rotation
displacementPerPulse := displacementPerRotation * rotationsPerPulse;

resetPulse(IN:= , PT:= resetWidth, Q=> clear, ET=> ); //reset pulse

IF NOT enable AND NOT AtInnerLimit THEN
	homingComplete := FALSE;
	step := Homing.IDLE;
	mode := HOLD;
END_IF

override();

CASE mode OF		
	HOLD: //hold current position, no motion
		pulse := 0;
		pulseRequest := 0;
	
	TARGET:	//target a given position
		
		IF WithinTolerance(position, targetPos, displacementPerPulse) THEN
			pulseRequest := 0;
			pulse := 0;
			mode := HOLD;
			
		ELSIF NOT Active THEN
			A :=  position < targetPos;
			(*
			2 options to traverse to a target position:
				a)  send all pulses at once - continuous motion but may exceed limits, check for bounds before setting
				b)  1 pulse at a time - choppy but safer
			*)
			targetPos := MAX(targetPos, minPosition); //if below minPosition, set to minPosition
			targetPos := MIN(targetPos, maxPosition); //if above maxPosition, set to maxPosition
			
			pulseRequest := TO_INT(ABS(position - targetPos)/displacementPerPulse);
			//pulseRequest := 1;
		END_IF
		
	CONTINUOUS: //single pulses in the direction specified by moveContinuous()
		pulseRequest := 1;
		
	RESET_ERR: //reset pulse, servo may need to be rehomed aftewards
		pulse := 0;
		pulseRequest := 0;
		resetPulse.IN := TRUE;
		
		IF resetPulse.Q THEN
			resetPulse.IN := FALSE;
			mode := HOLD;
		END_IF
		
END_CASE

sequence();

PROPERTY Active : BOOL
GET
Active := hlfb <> -9999;
END_GET
END_PROPERTY

{attribute 'monitoring':='call'}
PROPERTY AtOuterLimit : BOOL
GET
AtOuterLimit := outerLimit <> limitSensorDefaultState;
END_GET
END_PROPERTY

METHOD PRIVATE calculatePositions : BOOL
(*
the purpose of this method is calculate the position at the outer limit

complete a full range traverse while counting the pulses, then multiply
	displacement per rotation
	rotations per pulse
	number of pulses for the traversal
and add to position at inner limit to get position at outer limit
*)
CASE calculation OF
	IDLE:
		calculation := DOWN;
		
	DOWN:
		moveContinuous(direction := MC_Negative_Direction);
		IF AtInnerLimit THEN
			calculation := UP;
			pulseCounter := 0;
		END_IF
		
	UP:
		moveContinuous(direction := MC_Positive_Direction);
		IF AtHome THEN
			maxPosition := minPosition + (displacementPerRotation * rotationsPerPulse * pulseCounter);
			calculation := DONE;
		END_IF
		
	DONE:
		calculation := 0;
		calculatePositions := TRUE;
		
END_CASE
END_METHOD

PROPERTY CurrentPosition : LREAL
GET
CurrentPosition := position;

//CurrentPosition := pulsePosition * displacementPerPulse;
END_GET
SET
position := CurrentPosition;
END_SET
END_PROPERTY

PROPERTY Error : BOOL
GET
END_GET
END_PROPERTY

METHOD homingSequence : BOOL
homingDelay(IN:= , PT:= delayWidth, Q=> , ET=> );

CASE step OF
	Homing.IDLE:
		enable := TRUE;
		A := FALSE;
		B := TRUE;
		brakeRelease := TRUE;
		
		homingComplete := FALSE;
		
		homingDelay.IN := TRUE;
		IF homingDelay.Q THEN
			homingDelay.IN := FALSE;
			//step := Homing.START;
			step := Homing.RETRY;
		END_IF
		
	Homing.START:
		IF homingDelay.Q THEN
			homingDelay.IN := FALSE;
			step := Homing.SET;
			
		ELSIF AtHome THEN
			homingDelay.IN := TRUE;
			
		ELSIF AtOuterLimit THEN
			step := Homing.RETRY;
		
		ELSE
			enable := TRUE;
			A := FALSE;
			B := TRUE;
			brakeRelease := TRUE;
		
		END_IF
	
	Homing.RETRY:
		IF AtInnerLimit THEN
			homingDelay.IN := TRUE;
			enable := FALSE;
			
			IF homingDelay.Q THEN
				homingDelay.IN := FALSE;
				step := Homing.START;
			END_IF
			
		ELSE
			enable := TRUE;
			A := FALSE;
			B := FALSE;
			brakeRelease := TRUE;
			
			mode := CONTINUOUS;
		END_IF

	Homing.SET:
		enable := TRUE;
		A := FALSE;
		B := FALSE;
		brakeRelease := TRUE;
		
		IF calculatePositions() THEN
			step := Homing.DONE;
		END_IF
		
	Homing.DONE:
		homingSequence := homingComplete := TRUE;
		
		pulsePosition := 0;
		
		mode := HOLD;
		step := Homing.IDLE;
	
END_CASE
END_METHOD

{attribute 'TcRpcEnable'}
METHOD moveAbsolute : BOOL
VAR_INPUT
	newTarget : LREAL;
END_VAR
IF target >= maxPosition AND target <= minPosition THEN
	A :=  position < targetPos;
	targetPos := newTarget;
	mode := TARGET;
	
	moveAbsolute := TRUE;
END_IF
END_METHOD

{attribute 'TcRpcEnable'}
METHOD moveContinuous : BOOL
VAR_INPUT
	direction : MC_Direction;
END_VAR
IF direction = MC_Negative_Direction THEN
	A := FALSE;
ELSIF direction = MC_Positive_Direction THEN
	A := TRUE;
END_IF

mode := CONTINUOUS;
END_METHOD

{attribute 'TcRpcEnable'}
METHOD moveRelative : BOOL
VAR_INPUT
	distance : LREAL;
END_VAR
targetPos := targetPos + distance;

mode := TARGET;
END_METHOD

METHOD PRIVATE override : BOOL
VAR_INPUT
END_VAR
(*
allowable motion is between AtHome and AtInnerLimit
*)
IF AtHome AND NOT Active THEN
	IF homingDirectionOut THEN //homing is outwards
		position := maxPosition;
		pulsePosition := pulseCounter;
	ELSE
		position := minPosition;
		pulsePosition := 0;
	END_IF
	

ELSIF AtInnerLimit AND NOT Active THEN
	IF homingDirectionOut THEN //homing is outwards
		position := minPosition;
		pulsePosition := 0;
	ELSE
		position := maxPosition;
		pulsePosition := pulseCounter;
	END_IF
END_IF

CASE mode OF		
	HOLD:
		//
	
	TARGET:
		IF
			(AtHome AND TargetPosition > CurrentPosition) OR
			(AtInnerLimit AND TargetPosition > CurrentPosition) OR
			(AtOuterLimit AND TargetPosition < CurrentPosition)
		THEN
			mode := HOLD;
		END_IF
		
	CONTINUOUS:
		IF
			(AtHome AND A) OR
			(AtInnerLimit AND A) OR
			(AtOuterLimit AND NOT A)
		THEN
			mode := HOLD;
		END_IF
		
	RESET_ERR:
		//
		
END_CASE
END_METHOD

METHOD reset : BOOL
VAR_INPUT
END_VAR
mode := RESET_ERR;
END_METHOD

METHOD PRIVATE sequence : BOOL
VAR_INPUT
END_VAR
IF Active THEN //servo is active
	IF A THEN //positive direction
		position := position + (displacementPerPulse * pulse);
		pulsePosition := pulsePosition + pulse;
		
		pulseCounter := pulseCounter + pulse;
	ELSE //negative direction
		position := position - (displacementPerPulse * pulse);
		pulsePosition := pulsePosition - pulse;
		
		pulseCounter := pulseCounter - pulse;
	END_IF
	pulse := 0; //pulses already received, can be set to 0 so position change is not compounded

ELSIF pulse = 0 THEN //servo is not active
	pulse := pulseRequest;
END_IF

pulseRequest := 0; //remove this if not working as intended
END_METHOD

METHOD stop : BOOL
VAR_INPUT
END_VAR
mode := HOLD;
END_METHOD

PROPERTY TargetPosition : LREAL
GET
END_GET
SET
targetPos := TargetPosition;
END_SET
END_PROPERTY

METHOD toHome : BOOL
VAR_INPUT
END_VAR
IF homingDirectionOut THEN
	moveAbsolute(newTarget := maxPosition);
ELSE
	moveAbsolute(newTarget := minPosition);
END_IF
END_METHOD

END_FUNCTION_BLOCK

// ---- DUTs/Hardware/Insertion Package/Insertion.TcPOU
FUNCTION_BLOCK Insertion //2d insertion that combines a slider (alignment) and screw (push)
VAR_INPUT //interface references to existing drives
	slider : I_EncodedDrive;
	screw : I_ContinuousDrive;
END_VAR
VAR_OUTPUT
	contact AT %I* : BOOL;
	
	active : BOOL;
	error : BOOL;
	home : BOOL;
	
	homingComplete : BOOL;
	
	sliderPos : LREAL;
END_VAR
(*
this FB encapsulates 2 drives into a generic insertion machine
both drives should be declared externally in Hardware GVL as a concrete FB
Insertion instance should be declared and called in module scope, with the drives from Hardware GVL passed in by Interface reference
*)

homingComplete := slider.HomeSet AND screw.HomeSet;

active := slider.Active OR screw.Active;
error := slider.Error OR screw.Error;
home := slider.AtHome AND screw.AtHome;

sliderPos := slider.CurrentPosition;

METHOD align : BOOL
VAR_INPUT
	targetPos : REAL;
END_VAR
slider.moveAbsolute(newTarget := targetPos);
END_METHOD

METHOD homingSequence : BOOL
VAR_INPUT
END_VAR
IF NOT slider.homeSet THEN
	slider.homingSequence();
END_IF

IF NOT screw.homeSet THEN
	screw.homingSequence();
END_IF

homingSequence := homingComplete;
END_METHOD

METHOD press : BOOL
VAR_INPUT
END_VAR
screw.moveContinuous(direction := MC_Negative_Direction);
END_METHOD

METHOD release : BOOL
VAR_INPUT
END_VAR
screw.moveContinuous(direction := MC_Positive_Direction);
END_METHOD

METHOD reset : BOOL
VAR_INPUT
END_VAR
slider.reset();
screw.reset();
END_METHOD

METHOD stop : BOOL
VAR_INPUT
END_VAR
screw.stop();
slider.stop();
END_METHOD

METHOD toHome : BOOL
VAR_INPUT
END_VAR
slider.toHome();
screw.toHome();

toHome := slider.AtHome AND screw.AtHome;
END_METHOD

METHOD traverse : BOOL
VAR_INPUT
	direction : MC_Direction;
END_VAR
slider.moveContinuous(direction := MC_Negative_Direction);
END_METHOD

END_FUNCTION_BLOCK

// ---- DUTs/Hardware/Material Holders/StagingTable.TcPOU
FUNCTION_BLOCK StagingTable EXTENDS MaterialHolder

SUPER^();

METHOD autofill : BOOL
VAR_INPUT
	material : STRING;
END_VAR
VAR
	i : INT;
	slot : INT;
END_VAR
(*
this method will automatically find an open slot
*)
IF isFull() OR material = '' THEN
	RETURN;
END_IF

IF findOpenSlot(material := material, openSlot=> slot) THEN
	place(slot, material);
	autofill := TRUE;
END_IF
END_METHOD

METHOD findOpenSlot : BOOL
VAR_INPUT
	material : STRING;
END_VAR
VAR_OUTPUT
	openSlot : INT := 0;
END_VAR
VAR
	i : INT;
END_VAR
IF FIND(material, 'WDW') > 0 THEN //top wide, load in slot 9-10
	FOR i:=9 TO 10 BY 1 DO
		IF slots[i].material = '' THEN
			findOpenSlot := TRUE;
			openSlot := i;
			RETURN;
		END_IF
	END_FOR
	
ELSIF FIND(material, 'WD') > 0 THEN //standard width, load in slot 1-8
	FOR i:=1 TO 8 BY 1 DO
		IF slots[i].material = '' THEN
			findOpenSlot := TRUE;
			openSlot := i;
			RETURN;
		END_IF
	END_FOR
	
END_IF
END_METHOD

METHOD isEmpty : BOOL
VAR
	i : INT;
	temp : BOOL;
END_VAR
FOR i:=1 TO numSlots BY 1 DO
	temp := temp OR slots[i].occupied; //TRUE if any slots are occupied
END_FOR

isEmpty := NOT temp; //invert result - FALSE if any slots are occupied
END_METHOD

METHOD isFull : BOOL
VAR
	i : INT;
	temp : BOOL := TRUE;
END_VAR
FOR i:=1 TO numSlots BY 1 DO
	temp := temp AND slots[i].occupied;
END_FOR

isFull := temp;
END_METHOD

METHOD place : BOOL
VAR_INPUT
	i : INT;
	materialID : STRING;
END_VAR
IF slots[i].material = '' THEN
	slots[i].material := materialID;
	place := TRUE;
END_IF
END_METHOD

METHOD remove : BOOL
VAR_INPUT
	i : INT;
END_VAR
VAR_OUTPUT
	material : STRING;
END_VAR
remove := slots[i].material <> '';

material := slots[i].material;
slots[i].material := '';
END_METHOD

END_FUNCTION_BLOCK

// ---- DUTs/Hardware/Robots/KukaRobot.TcPOU
FUNCTION_BLOCK KukaRobot
VAR_OUTPUT
	forceStop AT %Q* : BOOL;
	resetSignal AT %Q* : BOOL;
	
	reservation : INT := SectionEnum.NULL_SECTION;
	
	error : BOOL;
	errId : DINT;
	
	outputs AT %Q* : ARRAY[1..50] OF WORD;
	inputs AT %I* : ARRAY[1..20] OF WORD;
END_VAR
VAR
	heartbeat : Watchdog;
	
	offline AT %I* : BOOL;
	toggleBit AT %I* : BOOL;
	
	hmiReservation : STRING;
END_VAR
(*
generic KUKA robot with 20 WORD outputs and 20 WORD inputs, connected to Beckhoff IPC via EL6692 or EL6695 EtherCAT bridge
includes minimal diagnostics to detect if robot is offline
robots should always be reserved before sending a task
*)

heartbeat(
	enable:= NOT offline,
	toggleBit:= toggleBit,
	timeoutWidth:= T#200MS,
	timeout=> );

error := //add any addition conditions with OR
	offline OR
	heartbeat.timeout;

//{attribute 'monitoring' := 'variable'}
{attribute 'monitoring' := 'call'}
PROPERTY Busy : BOOL
GET
END_GET
END_PROPERTY

METHOD clearCommand : BOOL
VAR_INPUT
END_VAR
MEMSET(ADR(outputs), 0, SIZEOF(outputs));
END_METHOD

//{attribute 'monitoring' := 'variable'}
{attribute 'monitoring' := 'call'}
PROPERTY Done : BOOL
GET
END_GET
END_PROPERTY

METHOD eStop : BOOL
VAR_INPUT
END_VAR
forceStop := TRUE;
eStop := TRUE;
END_METHOD

METHOD fullCommand : BOOL
VAR_INPUT
	newOutputs : REFERENCE TO ARRAY[1..50] OF WORD;
END_VAR
//IF NOT Busy THEN
	//RETURN;
//END_IF

outputs := newOutputs;
fullCommand := Done;

(*
CASE step OF
	SEND_COMMAND: //wait 1 cycle
		outputs := newOutputs;
		step := WAIT;
		
	WAIT:
		IF done THEN
			(*	
			IF NOT reset() THEN
				RETURN;
			END_IF
			
			step := 0;
			*)
			setCommandAndWait := TRUE;
		END_IF
		
END_CASE
*)
END_METHOD

{attribute 'monitoring' := 'call'}
PROPERTY Ready : BOOL
GET
END_GET
END_PROPERTY

METHOD release : BOOL
VAR_INPUT
	sectionReservation : SectionEnum;
END_VAR
IF reservation = sectionReservation THEN
	reservation := SectionEnum.NULL_SECTION;
	release := TRUE;
END_IF
END_METHOD

METHOD reserve : BOOL
VAR_INPUT
	reserveRequest : SectionEnum;
END_VAR
(*
this method exists because chipboard and wood bunk operations use the same robot
both sections need to check if the robot is open to commands before use
*)
IF Reserved AND reservation = reserveRequest THEN
	reserve := TRUE;

ELSIF NOT Reserved THEN
	reservation := reserveRequest;
	reserve := TRUE;

END_IF
END_METHOD

{attribute 'monitoring' := 'call'}
PROPERTY Reserved : BOOL
GET
Reserved := reservation <> SectionEnum.NULL_SECTION;
END_GET
END_PROPERTY

METHOD reset : BOOL
//resetSignal := TRUE;
//done := FALSE;

MEMSET(ADR(outputs), 0, SIZEOF(outputs));
(*
IF ready AND completedTask = 0 THEN
	resetSignal := FALSE;
	reset := TRUE;
END_IF
*)
END_METHOD

METHOD resume : BOOL
VAR_INPUT
END_VAR
forceStop := FALSE;

resume := NOT error AND errId = 0;
END_METHOD

METHOD setGroup : BOOL
VAR_INPUT
	group : INT;
	value : INT;
END_VAR
{warning disable C0195}
outputs[group] := value;
END_METHOD

END_FUNCTION_BLOCK

// ---- DUTs/Watchdog.TcPOU
FUNCTION_BLOCK Watchdog
VAR_INPUT
	enable : BOOL := TRUE; //watchdog can be disabled if needed
	
	toggleBit : BOOL;
	timeoutWidth : TIME := DEFAULT_ADS_TIMEOUT;
END_VAR
VAR_OUTPUT
	timeout : BOOL;
END_VAR
VAR	
	timer : TON;
	memoryBit : BOOL;
END_VAR

timer(
	IN:= enable AND (memoryBit = toggleBit), 
	PT:= timeoutWidth, 
	Q=> timeout, 
	ET=> );
	
(*
mem		tgbt	timer.IN
0		0		1
0		1		0
1		0		0
1		1		1
*)

END_FUNCTION_BLOCK

// ---- DUTs/Hardware/Robots/RobotA26.TcPOU
FUNCTION_BLOCK RobotA26 EXTENDS KukaRobot
VAR_INPUT
	conveyorSafety : BOOL;
END_VAR
VAR_OUTPUT //from outputs array
	{warning disable C0195}
	taskID : TaskA26;
	param1 : INT; //position number (1..6)
	param2 : INT;
	
	strapSafetyOut : BOOL;
END_VAR
VAR_OUTPUT //from inputs array
	tool : SectionEnum := SectionEnum.WOOD_BUNK;
	suspendedMaterial : STRING;
	
	completedTask : TaskA26;
	eoatDistance : INT;
	
	conveyorSafetyIn : BOOL;
END_VAR
VAR
	reservationEnum : SectionEnum;
	hmiTask : STRING;
	hmiTool : STRING;
END_VAR
(*
extends KukaRobot
	assigns descriptive labels to each IO group from the array
	additional section-specific methods to get/set IO groups
*)

(*
parameters - aliases to IO elements
command - full IO array
*)
{warning disable C0195}
SUPER^();

outputs[1] := taskID;
outputs[2] := param1;
outputs[3] := param2;

outputs[8].15 := conveyorSafety;

refreshParameters();

reservationEnum := reservation;
IF reservationEnum = SectionEnum.NULL_SECTION THEN
	hmiReservation := 'N/A';
ELSE
	hmiReservation := TO_STRING(reservationEnum);
END_IF

hmiTask := TO_STRING(taskID);
hmiTool := TO_STRING(tool);

{attribute 'monitoring' := 'call'}
PROPERTY Busy : BOOL
GET
VAR
	//emptyOutput : ARRAY[1..50] OF INT;
END_VAR
//Busy stays TRUE until outputs are cleared AND completed task has elapsed
//Ready is always inverse of Busy
refreshParameters();

Busy := taskID <> 0 OR completedTask <> 0;
END_GET
END_PROPERTY

METHOD clearCommand : BOOL
VAR_INPUT
END_VAR
SUPER^.clearCommand();

refreshParameters();
END_METHOD

{attribute 'monitoring' := 'call'}
PROPERTY Done : BOOL
GET
refreshParameters();

Done :=
	completedTask = taskID AND
	taskID <> 0 AND
	completedTask <> 0;
END_GET
END_PROPERTY

{attribute 'monitoring' := 'call'}
PROPERTY HoldMaterial : STRING
GET
HoldMaterial := suspendedMaterial;
END_GET
SET
suspendedMaterial := HoldMaterial;
END_SET
END_PROPERTY

{attribute 'monitoring' := 'call'}
PROPERTY Ready : BOOL
GET
refreshParameters();

Ready := taskID = 0 AND completedTask = 0;
END_GET
END_PROPERTY

METHOD PRIVATE refreshParameters : BOOL
VAR_INPUT
END_VAR
{warning disable C0196}
taskID := outputs[1];
param1 := outputs[2];
param2 := outputs[3];

conveyorSafetyIn := inputs[4].15;
END_METHOD

METHOD setGroup : BOOL
VAR_INPUT
	group : INT;
	value : INT;
END_VAR
SUPER^.setGroup(group := group, value := value);

refreshParameters();
END_METHOD

METHOD setParameters : BOOL
VAR_INPUT
	newTaskID : INT;
	newParam1 : INT;
	newParam2 : INT;
	newXmm : INT;
	newYmm : INT;
	newZmm : INT;
	newAngle : INT;
	newStagingOccupancy : INT;
	newInsertionSuctionStatus : INT;
	newMagazineStatus : INT; //unused
	newInspectionValue : INT;
END_VAR
VAR_INPUT
	strapSafety : BOOL;
END_VAR
setGroup(group := 1, value := newTaskID);
setGroup(group := 2, value := newParam1);
setGroup(group := 3, value := newParam2);

refreshParameters();
END_METHOD

END_FUNCTION_BLOCK

// ---- DUTs/Containers/PtrQueue.TcPOU
FUNCTION_BLOCK PtrQueue EXTENDS Queue //stores pointers to bundles, not the bundles themselves
VAR_INPUT
	
END_VAR
VAR
	elements : FB_BA_DynamicArray := (uiEntrySize := SIZEOF(PVOID), uiMinExpCount := Consts.initArraySize);
	//length : USINT := 0;
END_VAR

METHOD get : PVOID;
VAR_INPUT
	i : UINT;
END_VAR
elements.GetEntry(diIndex := i, pResultEntry := ADR(get));
END_METHOD

METHOD isEmpty : BOOL
VAR_INPUT
END_VAR
isEmpty := (elements.diCount = 0);
END_METHOD

METHOD poll : PVOID;
VAR_INST
	i : UINT;
END_VAR
poll := get(i := 0);
elements.RemoveEntry(diIndex := 0);
//length := length - 1;
END_METHOD

METHOD push : BOOL
VAR_INPUT
	value : PVOID;
END_VAR
elements.AddEntryPtr(pEntry := value);
//length := length + 1;
push := TRUE;
END_METHOD

METHOD size : DINT
VAR_INPUT
END_VAR
size := elements.diCount;
END_METHOD

END_FUNCTION_BLOCK

// ---- DUTs/Containers/IntQueue.TcPOU
FUNCTION_BLOCK IntQueue EXTENDS Queue
VAR
	elements : FB_BA_DynamicArray := (uiEntrySize := SIZEOF(INT), uiMinExpCount := CONSTS.initArraySize);
	//length : USINT := 0;
END_VAR

METHOD clear : BOOL
VAR_INPUT
END_VAR
elements.Reset();
length := 0;
END_METHOD

METHOD contains : BOOL
VAR_INPUT
	value : INT;
END_VAR
VAR
	temp : INT;
	i : INT;
END_VAR
IF length = 0 THEN
	contains := FALSE;
	RETURN;
END_IF

FOR i:=0 TO (length-1) BY 1 DO
	temp := get(i);
	IF MEMCMP(ADR(temp), ADR(value), SIZEOF(INT)) = 0 THEN
		contains := TRUE;
		RETURN;
	END_IF
END_FOR
contains := FALSE;
END_METHOD

METHOD get : INT
VAR_INPUT
	i : INT;
END_VAR
elements.GetEntry(diIndex := i, pResultEntry := ADR(get));
END_METHOD

METHOD isEmpty : BOOL
VAR_INPUT
END_VAR
isEmpty := (elements.diCount = 0);
END_METHOD

METHOD poll : INT
VAR_INST
	temp : INT;
	i : UINT;
END_VAR
temp := get(i := 0);
elements.RemoveEntry(diIndex := 0);
//length := length - 1;
poll := temp;
END_METHOD

METHOD push : BOOL
VAR_INPUT
	value : INT;
END_VAR
elements.AddEntry(pEntry := ADR(value));
//length := length + 1;
END_METHOD

METHOD set : BOOL
VAR_INPUT
	i : INT;
	value : INT;
END_VAR
IF i > 0 AND i < length THEN
	elements.SetEntry(i, ADR(value));
	set := TRUE;
END_IF
END_METHOD

METHOD size : DINT
VAR_INPUT
END_VAR
size := elements.diCount;
END_METHOD

END_FUNCTION_BLOCK

// ---- DUTs/Containers/StringQueue.TcPOU
FUNCTION_BLOCK StringQueue EXTENDS Queue
VAR
	elements : FB_BA_DynamicArray := (uiEntrySize := SIZEOF(STRING), uiMinExpCount := CONSTS.initArraySize);
	//length : USINT := 0;
END_VAR

METHOD get : STRING
VAR_INPUT
	i : UINT;
END_VAR
elements.GetEntry(diIndex := i, pResultEntry := ADR(get));
END_METHOD

METHOD isEmpty : BOOL
VAR_INPUT
END_VAR
isEmpty := (elements.diCount = 0);
END_METHOD

METHOD poll : STRING
VAR_INST
	temp : STRING;
	i : UINT;
END_VAR
temp := get(i := 0);
elements.RemoveEntry(diIndex := 0);
//length := length - 1;
poll := temp;
END_METHOD

METHOD push : BOOL
VAR_INPUT
	value : STRING;
END_VAR
elements.AddEntry(pEntry := ADR(value));
//length := length + 1;
END_METHOD

METHOD size : DINT
VAR_INPUT
END_VAR
size := elements.diCount;
END_METHOD

END_FUNCTION_BLOCK

// ---- HARDWARE_DISTRUBUTION/ConveyorControlModule.TcPOU
PROGRAM ConveyorControlModule
VAR_IN_OUT
	A24_LRC_C02 	: Conveyor; //these conveyoors move bundles from A2.7 to A2.4
	A24_LRC_C04 	: Conveyor;
	A24_LRC_C06	 	: Conveyor;
	A24_LRC_C08 	: Conveyor;
	A24_LRC_C10 	: Conveyor;
	A24_LRC_C12 	: Conveyor;
	
	A24_SC_C01 		: ConveyorSC; //these conveyors move bundles on A2.4 forward down the cell
	A24_SC_C03 		: ConveyorSC;
	A24_SC_C05 		: ConveyorSC;
	A24_SC_C07 		: ConveyorSC;
	A24_SC_C09 		: ConveyorSC;
	A24_SC_C11 		: ConveyorSC;
	A24_SC_C13 		: ConveyorSC;
	
	A23_LSC_C14 	: ConveyorLSC;
	
	A22_SC_C15 		: ConveyorSC;
	A22_LSC_C16 	: ConveyorLSC;
	A22_LSC_C17 	: ConveyorLSC;
	
	A21_SC_C18 		: ConveyorSC;
	A21_LSC_C19 	: ConveyorLSC;
	A21_LSC_C20 	: ConveyorLSC;
	A21_LSC_C21 	: ConveyorLSC;
	
	A25_SC_C22 		: ConveyorSC;
	A25_SC_C24 		: ConveyorSC;
	A25_SC_C26 		: ConveyorSC;
	A25_SC_C28 		: ConveyorSC;
	A25_SC_C30 		: ConveyorSC;
	
	A25_LSC_C23 	: ConveyorLSC; //these conveyors move the bundle sideways onto the output buffers
	A25_LSLCC_C25 	: ConveyorLSC;
	A25_LSLCC_C27 	: ConveyorLSC;
	A25_LSC_C29 	: ConveyorLSC;
	A25_SC_C31 		: ConveyorSC;
	A25_SC_C32 		: ConveyorSC;
	A25_SC_C33 		: ConveyorSC;
	A25_SC_C34 		: ConveyorSC;
	A25_SC_C35 		: ConveyorSC;
	A25_SC_C36 		: ConveyorSC;
	A25_SC_C37 		: ConveyorSC;
	A25_SC_C38 		: ConveyorSC;
END_VAR
VAR
	conveyorsArr : ARRAY[1..38] OF POINTER TO ConveyorSC;
	
	spoolTimer : TON;
	i : DINT := 1;
END_VAR
VAR CONSTANT
	spoolSpacing : TIME := T#100MS;
END_VAR

pushConveyorsToArray();
linkCompute();

spoolTimer(IN:= , PT:= spoolSpacing, Q=> , ET=> );
spoolTimer.IN := TRUE;

IF
	(conveyorsArr[i]^.requestedMode = ConveyorMode.FORWARD OR conveyorsArr[i]^.requestedMode = ConveyorMode.BACKWARD) AND //conveyor requests motion
	conveyorsArr[i]^.requestedMode <> conveyorsArr[i]^.trueMode AND //conveyor request differs from current operation
	spoolTimer.Q //ready to spool
THEN
	//spool up conveyor
	i := (i + 1) MOD (CONSTS.numCellConveyors + 1) + 1;
	spoolTimer.IN := FALSE;
END_IF

METHOD PRIVATE linkCompute : BOOL
VAR
	i : DINT;
	j : DINT;
	
	linkStart : DINT := -1;
	linkEnd : DINT := -1;
	
	priorityInLink : ConveyorMode;
END_VAR
(*
link interation method 
slower, but will correctly set all operations every cycle
*)
FOR i:=1 TO CONSTS.numCellConveyors BY 1 DO
	IF conveyorsArr[i]^.IsOccupied THEN
		
		IF linkStart = -1 THEN
			linkStart := i;
		END_IF
		
		priorityInLink := MAX(priorityInLink, conveyorsArr[i]^.requestedMode);
		linkEnd := i;
		
	ELSIF linkStart <> -1 AND linkEnd <> -1 THEN //set all conveyor operations to priorityInLink
		linkEnd := i-1;
		
		FOR j:=linkStart TO linkEnd BY 1 DO
			conveyorsArr[j]^.setMode(priorityInLink);
		END_FOR
		
		linkStart := -1;
		linkEnd := -1;
		priorityInLink := ConveyorMode.IDLE;
		
		CONTINUE;
	END_IF
	
END_FOR

IF linkStart > -1 AND linkEnd > -1 THEN
	FOR j:=linkStart TO linkEnd BY 1 DO
		conveyorsArr[j]^.setMode(priorityInLink);
	END_FOR
END_IF
END_METHOD

METHOD PRIVATE pushConveyorsToArray : BOOL
{warning disable C0371}
conveyorsArr[1] := ADR(A24_SC_C01);
conveyorsArr[2] := ADR(A24_LRC_C02);
conveyorsArr[3] := ADR(A24_SC_C03);
conveyorsArr[4] := ADR(A24_LRC_C04);
conveyorsArr[5] := ADR(A24_SC_C05);
conveyorsArr[6] := ADR(A24_LRC_C06);
conveyorsArr[7] := ADR(A24_SC_C07);
conveyorsArr[8] := ADR(A24_LRC_C08);
conveyorsArr[9] := ADR(A24_SC_C09);
conveyorsArr[10] := ADR(A24_LRC_C10);
conveyorsArr[11] := ADR(A24_SC_C11);
conveyorsArr[12] := ADR(A24_LRC_C12);
conveyorsArr[13] := ADR(A24_SC_C13);

conveyorsArr[14] := ADR(A23_LSC_C14);

conveyorsArr[15] := ADR(A22_SC_C15);
conveyorsArr[16] := ADR(A22_LSC_C16);
conveyorsArr[17] := ADR(A22_LSC_C17);

conveyorsArr[18] := ADR(A21_SC_C18);
conveyorsArr[19] := ADR(A21_LSC_C19);
conveyorsArr[20] := ADR(A21_LSC_C20);
conveyorsArr[21] := ADR(A21_LSC_C21);

conveyorsArr[22] := ADR(A25_SC_C22);
conveyorsArr[23] := ADR(A25_LSC_C23);
conveyorsArr[24] := ADR(A25_SC_C24);
conveyorsArr[25] := ADR(A25_LSLCC_C25);
conveyorsArr[26] := ADR(A25_SC_C26);
conveyorsArr[27] := ADR(A25_LSLCC_C27);
conveyorsArr[28] := ADR(A25_SC_C28);
conveyorsArr[29] := ADR(A25_LSC_C29);
conveyorsArr[30] := ADR(A25_SC_C30);
conveyorsArr[31] := ADR(A25_SC_C31);
conveyorsArr[32] := ADR(A25_SC_C32);
conveyorsArr[33] := ADR(A25_SC_C33);
conveyorsArr[34] := ADR(A25_SC_C34);
conveyorsArr[35] := ADR(A25_SC_C35);
conveyorsArr[36] := ADR(A25_SC_C36);
conveyorsArr[37] := ADR(A25_SC_C37);
conveyorsArr[38] := ADR(A25_SC_C38);
END_METHOD

END_PROGRAM

// ---- HARDWARE_DISTRUBUTION/ConveyorSyncUnit.TcPOU
PROGRAM ConveyorSyncUnit
VAR_OUTPUT
	A24_LRC_C02 	: Conveyor; //these conveyoors move bundles from A2.7 to A2.4
	A24_LRC_C04 	: Conveyor;
	A24_LRC_C06	 	: Conveyor;
	A24_LRC_C08 	: Conveyor;
	A24_LRC_C10 	: Conveyor;
	A24_LRC_C12 	: Conveyor;
	
	A24_SC_C01 		: ConveyorSC; //these conveyors move bundles on A2.4 forward down the cell
	A24_SC_C03 		: ConveyorSC;
	A24_SC_C05 		: ConveyorSC;
	A24_SC_C07 		: ConveyorSC;
	A24_SC_C09 		: ConveyorSC;
	A24_SC_C11 		: ConveyorSC;
	A24_SC_C13 		: ConveyorSC;
	
	A23_LSC_C14 	: ConveyorLSC;
	
	A22_SC_C15 		: ConveyorSC;
	A22_LSC_C16 	: ConveyorLSC;
	A22_LSC_C17 	: ConveyorLSC;
	
	A21_SC_C18 		: ConveyorSC;
	A21_LSC_C19 	: ConveyorLSC;
	A21_LSC_C20 	: ConveyorLSC;
	A21_LSC_C21 	: ConveyorLSC;
	
	A25_SC_C22 		: ConveyorSC;
	A25_SC_C24 		: ConveyorSC;
	A25_SC_C26 		: ConveyorSC;
	A25_SC_C28 		: ConveyorSC;
	A25_SC_C30 		: ConveyorSC;
	
	A25_LSC_C23 	: ConveyorLSC; //these conveyors move the bundle sideways onto the output buffers
	A25_LSLCC_C25 	: ConveyorLSC;
	A25_LSLCC_C27 	: ConveyorLSC;
	A25_LSC_C29 	: ConveyorLSC;
	A25_SC_C31 		: ConveyorSC;
	A25_SC_C32 		: ConveyorSC;
	A25_SC_C33 		: ConveyorSC;
	A25_SC_C34 		: ConveyorSC;
	A25_SC_C35 		: ConveyorSC;
	A25_SC_C36 		: ConveyorSC;
	A25_SC_C37 		: ConveyorSC;
	A25_SC_C38 		: ConveyorSC;
END_VAR
VAR
	conveyorsArr : ARRAY[1..38] OF POINTER TO ConveyorSC;
	
	spoolTimer : TON;
	i : DINT := 1;
END_VAR
VAR CONSTANT
	spoolSpacing : TIME := T#100MS;
END_VAR
(*
this module contains all conveyors, which can be used by subarea/section modules as required
*)

pushConveyorsToArray();
linkCompute();

spoolTimer(IN:= , PT:= spoolSpacing, Q=> , ET=> );
spoolTimer.IN := TRUE;

IF
	(conveyorsArr[i]^.requestedMode = ConveyorMode.FORWARD OR conveyorsArr[i]^.requestedMode = ConveyorMode.BACKWARD) AND //conveyor requests motion
	conveyorsArr[i]^.requestedMode <> conveyorsArr[i]^.trueMode AND //conveyor request differs from current operation
	spoolTimer.Q //ready to spool
THEN
	//spool up conveyor
	i := (i + 1) MOD (CONSTS.numCellConveyors + 1) + 1;
	spoolTimer.IN := FALSE;
END_IF

METHOD PRIVATE linkCompute : BOOL
VAR
	i : DINT;
	j : DINT;
	
	linkStart : DINT := -1;
	linkEnd : DINT := -1;
	
	priorityInLink : ConveyorMode;
END_VAR
(*
link interation method 
slower, but will correctly set all operations every cycle
*)
FOR i:=1 TO CONSTS.numCellConveyors BY 1 DO
	IF conveyorsArr[i]^.IsOccupied THEN
		
		IF linkStart = -1 THEN
			linkStart := i;
		END_IF
		
		priorityInLink := MAX(priorityInLink, conveyorsArr[i]^.requestedMode);
		linkEnd := i;
		
	ELSIF linkStart <> -1 AND linkEnd <> -1 THEN //set all conveyor operations to priorityInLink
		linkEnd := i-1;
		
		FOR j:=linkStart TO linkEnd BY 1 DO
			conveyorsArr[j]^.setMode(priorityInLink);
		END_FOR
		
		linkStart := -1;
		linkEnd := -1;
		priorityInLink := ConveyorMode.IDLE;
		
		CONTINUE;
	END_IF
	
END_FOR

IF linkStart > -1 AND linkEnd > -1 THEN
	FOR j:=linkStart TO linkEnd BY 1 DO
		conveyorsArr[j]^.setMode(priorityInLink);
	END_FOR
END_IF
END_METHOD

METHOD PRIVATE pushConveyorsToArray : BOOL
{warning disable C0371}
conveyorsArr[1] := ADR(A24_SC_C01);
conveyorsArr[2] := ADR(A24_LRC_C02);
conveyorsArr[3] := ADR(A24_SC_C03);
conveyorsArr[4] := ADR(A24_LRC_C04);
conveyorsArr[5] := ADR(A24_SC_C05);
conveyorsArr[6] := ADR(A24_LRC_C06);
conveyorsArr[7] := ADR(A24_SC_C07);
conveyorsArr[8] := ADR(A24_LRC_C08);
conveyorsArr[9] := ADR(A24_SC_C09);
conveyorsArr[10] := ADR(A24_LRC_C10);
conveyorsArr[11] := ADR(A24_SC_C11);
conveyorsArr[12] := ADR(A24_LRC_C12);
conveyorsArr[13] := ADR(A24_SC_C13);

conveyorsArr[14] := ADR(A23_LSC_C14);

conveyorsArr[15] := ADR(A22_SC_C15);
conveyorsArr[16] := ADR(A22_LSC_C16);
conveyorsArr[17] := ADR(A22_LSC_C17);

conveyorsArr[18] := ADR(A21_SC_C18);
conveyorsArr[19] := ADR(A21_LSC_C19);
conveyorsArr[20] := ADR(A21_LSC_C20);
conveyorsArr[21] := ADR(A21_LSC_C21);

conveyorsArr[22] := ADR(A25_SC_C22);
conveyorsArr[23] := ADR(A25_LSC_C23);
conveyorsArr[24] := ADR(A25_SC_C24);
conveyorsArr[25] := ADR(A25_LSLCC_C25);
conveyorsArr[26] := ADR(A25_SC_C26);
conveyorsArr[27] := ADR(A25_LSLCC_C27);
conveyorsArr[28] := ADR(A25_SC_C28);
conveyorsArr[29] := ADR(A25_LSC_C29);
conveyorsArr[30] := ADR(A25_SC_C30);
conveyorsArr[31] := ADR(A25_SC_C31);
conveyorsArr[32] := ADR(A25_SC_C32);
conveyorsArr[33] := ADR(A25_SC_C33);
conveyorsArr[34] := ADR(A25_SC_C34);
conveyorsArr[35] := ADR(A25_SC_C35);
conveyorsArr[36] := ADR(A25_SC_C36);
conveyorsArr[37] := ADR(A25_SC_C37);
conveyorsArr[38] := ADR(A25_SC_C38);
END_METHOD

END_PROGRAM

// ---- POUs/Helper Functions/General/TimestructToString.TcPOU
FUNCTION TimestructToString : STRING
VAR_INPUT
	t : REFERENCE TO TIMESTRUCT;
END_VAR
VAR
	year : STRING;
	month : STRING;
	day : STRING;
	
	hour : STRING;
	minute : STRING;
	second : STRING;
	
	strIn : ARRAY[0..5] OF STRING(2);
	
	sCMD : STRING;
END_VAR

strIn[0] := WORD_TO_STRING(t.wYear);
strIn[1] := WORD_TO_STRING(t.wMonth);
strIn[2] := WORD_TO_STRING(t.wDay);

strIn[3] := WORD_TO_STRING(t.wHour);
strIn[4] := WORD_TO_STRING(t.wMinute);
strIn[5] := WORD_TO_STRING(t.wSecond);

sCMD := CONCAT(strIn[0], '-'); //date
sCMD := CONCAT(sCMD, strIn[1]);
sCMD := CONCAT(sCMD, '-');
sCMD := CONCAT(sCMD, strIn[2]);
sCMD := CONCAT(sCMD, ' ');

sCMD := CONCAT(sCMD, strIn[3]); //time
sCMD := CONCAT(sCMD, ':');
sCMD := CONCAT(sCMD, strIn[4]);
sCMD := CONCAT(sCMD, ':');
sCMD := CONCAT(sCMD, strIn[5]);

END_FUNCTION

// ---- POUs/Helper Functions/Hardware Modules/SetSuctions.TcPOU
FUNCTION SetSuctions : BOOL
VAR_IN_OUT
	suctions : ARRAY[*] OF SuctionPad;
END_VAR
VAR_INPUT
	state : BOOL;
END_VAR
VAR
	i : DINT;
END_VAR

FOR i:=LOWER_BOUND(suctions, 1) TO UPPER_BOUND(suctions, 1) BY 1 DO
	suctions[i].enable := state;
END_FOR

END_FUNCTION

// ---- POUs/Helper Functions/Hardware Modules/SetSuctionsPtr.TcPOU
FUNCTION SetSuctionsPtr : BOOL
VAR_INPUT
	suctions : POINTER TO SuctionPad;
	numPads : DINT;
	
	state : BOOL;
END_VAR
VAR
	i : DINT;
END_VAR

FOR i:=0 TO numPads-1 BY 1 DO
	suctions[i].enable := state;
END_FOR

END_FUNCTION

// ---- POUs/Helper Functions/Hardware Modules/SetupHardware.TcPOU
FUNCTION SetupHardware : BOOL
VAR
	iWoodBunkSlot : WoodBunk;
	iChipboardSlot : Chipboard;
	
	i : INT;
END_VAR

FOR iWoodBunkSlot:=1 TO WoodBunk.size-1 BY 1 DO //init wood bunk magazine slots
	magazineA21Left.setSlot(i := iWoodBunkSlot, material := TO_STRING(iWoodBunkSlot), error => );
	magazineA21Right.setSlot(i := iWoodBunkSlot, material := TO_STRING(iWoodBunkSlot), error => );
END_FOR

//--------------------------------------------------

FOR iChipboardSlot:=1 TO Chipboard.size-1 BY 1 DO //init chipboard skid slots
	skidA21Left.setSlot(i := iChipboardSlot, material := TO_STRING(iChipboardSlot), error => );
	skidA21Right.setSlot(i := iChipboardSlot, material := TO_STRING(iChipboardSlot), error => );
END_FOR

//--------------------------------------------------

FOR i:=1 TO CONSTS.maxQueue BY 1 DO //get wood bunk magazine + chipboard skid availability from robot1 and robot2
	{warning disable C0195}
	skidA21Left.setOccupancy( i := i, occupancy := IntegerBitAccess(robot1.inputs[4], i-1) );
	skidA21Right.setOccupancy( i := i, occupancy := IntegerBitAccess(robot2.inputs[4], i-1) );

	magazineA21Left.setOccupancy( i := i, occupancy := IntegerBitAccess(robot1.inputs[3], i-1) );
	magazineA21Right.setOccupancy( i := i, occupancy := IntegerBitAccess(robot2.inputs[3], i-1) );
END_FOR

//--------------------------------------------------

//enable all drives
verticalDriveA21Left.bEnable := TRUE;
verticalDriveA21Right.bEnable := TRUE;
insertionA21Left.enable := TRUE;
horizontalDriveA21Left.bEnable := TRUE;
horizontalDriveA21Right.bEnable := TRUE;
insertionA21Right.enable := TRUE;
pistonA21Bottom.bEnable := TRUE;

SetupHardware := TRUE;

END_FUNCTION

// ---- POUs/Helper Functions/Hardware Modules/SuctionQualityPtr.TcPOU
FUNCTION SuctionQualityPtr  : BOOL
VAR_INPUT
	suctions : POINTER TO SuctionPad;
	numPads : DINT;
END_VAR
VAR_INPUT
	insertionMaterial : STRING;
	recipeMaterial : STRING;
END_VAR
VAR
	i : DINT;
	
	failedVacuums : INT;
	numVacuums : INT;
END_VAR

(*
IF insertionMaterial <> recipeMaterial THEN //reintroduce this condition later
	RETURN;
END_IF
*)

FOR i:=0 TO numPads BY 1 DO
	IF suctions[i].enable THEN
		numVacuums := numVacuums + 1;
		IF NOT suctions[i].occupied THEN
			failedVacuums := failedVacuums + 1;
		END_IF
	END_IF
	
END_FOR

//SuctionQualityPtrArr := failedVacuums < (numVacuums * 1/3);
SuctionQualityPtr := TRUE;

END_FUNCTION

// ---- POUs/Helper Functions/Material Functions/GetPairMasterLength.TcPOU
FUNCTION GetPairMasterLength : LREAL
VAR_INPUT
	currentPair : REFERENCE TO PositionMaterials;
END_VAR
VAR
	topLength : LREAL;
	leftLength : LREAL;
	rightLength : LREAL;
	bottomLength : LREAL;
	
	topLeftLength : LREAL;
	topRightLength : LREAL;
	bottomLeftLength : LREAL;
	bottomRightLength : LREAL;
END_VAR

topLength := GetMaterialLength(currentPair.top);
leftLength := GetMaterialLength(currentPair.left);
rightLength := GetMaterialLength(currentPair.right);
bottomLength := GetMaterialLength(currentPair.bottom);

topLeftLength := GetMaterialLength(currentPair.topLeft);
topRightLength := GetMaterialLength(currentPair.topRight);
bottomLeftLength := GetMaterialLength(currentPair.bottomLeft);
bottomRightLength := GetMaterialLength(currentPair.bottomRight);

GetPairMasterLength := MAX(topLength, leftLength, rightLength, bottomLength, topLeftLength, topRightLength, bottomLeftLength, bottomRightLength);

END_FUNCTION

// ---- POUs/Helper Functions/Material Functions/GetMaterialLength.TcPOU
FUNCTION GetMaterialLength : LREAL
VAR_INPUT
	material : STRING;
END_VAR
VAR
	i : INT;
END_VAR

FOR i:=0 TO Consts.numMaterials BY 1 DO
	IF Consts.allMaterials[i].code = material THEN
		getMaterialLength := Consts.allMaterials[i].length;
		RETURN;
	END_IF
END_FOR
//otherwise, return 0
GetMaterialLength := 0;

END_FUNCTION

// ---- POUs/MAIN.TcPOU
PROGRAM MAIN
VAR_OUTPUT //globally readable, but only modifiable by MAIN
	outputBuffer : ARRAY[Surface.LEFT..Surface.RIGHT] OF Bundle;
	outputBufferPass, outputBufferFail : Bundle;
	numOutputBundles : USINT := 0;
	
	bundleIn : Bundle;
	bundleOut : Bundle;
	
	start : BOOL;
	
	ready : BOOL;
	busy : BOOL;
	done : BOOL;
	error : BOOL;
	backlog : BOOL;
	
	stop : BOOL;
	execute : BOOL;
	hold : BOOL;
	reset : BOOL;
	
	localTime : TIMESTRUCT;
	
	pmlModeString : STRING;
	pmlStateString : STRING;
END_VAR
VAR
	clearPassBuffer, clearFailBuffer AT %I* : BOOL;
	receiverStruct : AdsData;
	
	//ETA is not strictly required, area will process bundle even if it is not in ETA arrays
	expectedBundles : ARRAY[0..CONSTS.maxQueue] OF STRING; //bundles expected to arrive
	expectedArrivals : ARRAY[0..CONSTS.maxQueue] OF TIMESTRUCT; //bundles expected to arrive
	numEtaBundles : INT;
	
	//parallel arrays - bundle, bypass
	numBundles : INT;
	bundlesQueue : ARRAY[0..CONSTS.maxQueue] OF Bundle;
	bundlesBypass : ARRAY[0..CONSTS.maxQueue] OF BOOL;
END_VAR
VAR //sections
	spacerRecollector : SpacerRecollectionUnit;
	//paperSection : PaperEx;
	cardboardSection : CardboardEx;
	chipboardSection : ChipboardEx;
	woodBunkSection : WoodBunkEx;
	//outputSection : AreaOutputEx;	
END_VAR
VAR
	fbLocalSystemTime : FB_LocalSystemTime;
	dbLogger : SqlDatabaseAccessor;
	
	pmlState : E_PMLState;
	pmlCommand : E_PMLCommand;
	pmlStateMachine : PML_StateMachine;
	
	pmlModeRequest : E_PMLCustomUnitMode := ePMLCustomUnitMode_Production;
	pmlMode : E_PMLCustomUnitMode;
	pmlModeManager : PML_UnitModeManager;
END_VAR
VAR //these variables are only tracked for HMI
	sectionsBusy : ARRAY[0..SectionEnum.size] OF BOOL;
	sectionsIterator : ARRAY[0..SectionEnum.size] OF INT;
END_VAR

(*
ready := paperSection.ready; //if A2 is not ready, dispatch controller must block operator from sending bundles here
busy := paperSection.busy OR cardboardCornerGuardSection.busy OR chipboardSection.busy OR woodBunkSection.busy OR outputSection.busy;
done := outputSection.done;
backlog := numBundlesQueue > 5;
*)

initSections();

//for random testing only
//fillBundlesQueue();
//SizeCheck();

blocks();
	
runPML();

(*
the new program structure specifies the following:
	declare the section modules in MAIN,
	declare the hardware modules in the approrpiate subarea module
		see folder HARDWARE_DISTRIBUTION for all 6 subareas
	pass the section modules to one of the 6 subarea hardware distrubutors to be called with their required hardware

conveyors are declared as VAR_OUTPUTs to allow an external conveyor ocntrol module to access all conveyors across subareas

this structure should drastically reduce the visibility of hardware modules and eliminate the need for large GVLs
*)

A26(spacerRecollector := spacerRecollector);
(*
A24()
A23()
*)
A22(
	sectionCC:= cardboardSection,
	bundlesQueue:= bundlesQueue, 
	bundlesBypass:= bundlesBypass);
	
A21(
	sectionCIP:= chipboardSection, 
	sectionWB:= woodBunkSection, 
	bundlesQueue:= bundlesQueue, 
	bundlesBypass:= bundlesBypass);
//A25()

IF AdsClient.fetchData(receiverStruct) THEN
	interpretTransmission(receiverStruct);
END_IF

IF ready AND BundleIsValid(bundleIn) THEN
	receive();
END_IF

IF clearPassBuffer OR clearFailBuffer THEN
	transfer();
	shiftBundles();
END_IF

dbLogger();

METHOD PRIVATE blocks : BOOL
VAR_INPUT
END_VAR
fbLocalSystemTime(
	sNetID:= '', 
	bEnable:= TRUE, 
	dwCycle:= , 
	dwOpt:= , 
	tTimeout:= , 
	bValid=> , 
	systemTime=> localTime, 
	tzID=> );

ConveyorControlModule(
	A24_LRC_C02:= A24.A24_LRC_C02, 
	A24_LRC_C04:= A24.A24_LRC_C04, 
	A24_LRC_C06:= A24.A24_LRC_C06, 
	A24_LRC_C08:= A24.A24_LRC_C08, 
	A24_LRC_C10:= A24.A24_LRC_C10, 
	A24_LRC_C12:= A24.A24_LRC_C12, 
	
	A24_SC_C01:= A24.A24_SC_C01, 
	A24_SC_C03:= A24.A24_SC_C03, 
	A24_SC_C05:= A24.A24_SC_C05, 
	A24_SC_C07:= A24.A24_SC_C07, 
	A24_SC_C09:= A24.A24_SC_C09, 
	A24_SC_C11:= A24.A24_SC_C11, 
	A24_SC_C13:= A24.A24_SC_C13, 
	
	A23_LSC_C14:= A23.A23_LSC_C14, 
	
	A22_SC_C15:= A22.A22_SC_C15, 
	A22_LSC_C16:= A22.A22_LSC_C16, 
	A22_LSC_C17:= A22.A22_LSC_C17, 
	A21_SC_C18:= A21.A21_SC_C18, 
	A21_LSC_C19:= A21.A21_LSC_C19, 
	A21_LSC_C20:= A21.A21_LSC_C20, 
	A21_LSC_C21:= A21.A21_LSC_C21, 
	
	A25_SC_C22:= A25.A25_SC_C22, 
	A25_LSC_C23:= A25.A25_LSC_C23, 
	A25_SC_C24:= A25.A25_SC_C24, 
	A25_LSLCC_C25:= A25.A25_LSLCC_C25, 
	A25_SC_C26:= A25.A25_SC_C26, 
	A25_LSLCC_C27:= A25.A25_LSLCC_C27, 
	A25_SC_C28:= A25.A25_SC_C28, 
	A25_LSC_C29:= A25.A25_LSC_C29, 
	A25_SC_C30:= A25.A25_SC_C30, 
	
	
	A25_SC_C31:= A25.A25_SC_C31, 
	A25_SC_C32:= A25.A25_SC_C32, 
	A25_SC_C33:= A25.A25_SC_C33, 
	A25_SC_C34:= A25.A25_SC_C34, 
	A25_SC_C35:= A25.A25_SC_C35, 
	A25_SC_C36:= A25.A25_SC_C36, 
	A25_SC_C37:= A25.A25_SC_C37, 
	A25_SC_C38:= A25.A25_SC_C38);
	
AdsClient( //PLC-PLC comms
	ServerNetId:= , 
	ServerPort:= , 
	bBusy=> , 
	err=> , 
	errid=> , 
	localPrgName=> , 
	localNetId=> , 
	localPort=> , 
	socketReady=> , 
	remoteAccessPrefix=> );
	
TcpServer1Vision( //PLC-Vision comms
	ServerNetId:= , 
	ServerAdr:= , 
	ServerPort:= , 
	busy=> , 
	error=> , 
	errorId=> , 
	bytesReceived=> , 
	connected=> , 
	receiveStruct=> );
END_METHOD

METHOD fillBundlesQueue : BOOL
VAR
	i : INT;
END_VAR
IF NOT start THEN //for HMI testing only, remove for production
	FOR i:=0 TO CONSTS.maxQueue BY 1 DO
		bundlesQueue[i].id := TO_STRING(i);
	END_FOR
	
	start := TRUE;
END_IF
END_METHOD

METHOD PRIVATE initSections : BOOL
//paperSection.connectTo(ADR(cardboardCornerGuardSection));
//cardboardCornerGuardSection.connectTo(ADR(chipboardSection));
//chipboardSection.connectTo(ADR(woodBunkSection));
woodBunkSection.connectTo(0); //(ADR(outputSection));
//connecting to 0 means no next section

//paperSection.sectionID := SectionEnum.PAPER;
//cardboardCornerGuardSection.sectionID := SectionEnum.CARDBOARD_CORNERGUARD;
//chipboardSection.sectionID := SectionEnum.CHIPBOARD;
woodBunkSection.sectionID := SectionEnum.WOOD_BUNK;
//outputSection.sectionID := SectionEnum.OUTPUT;

(*
	paperSection.pNextSection := ADR(cardboardCornerGuardSection);
	cardboardCornerGuardSection.accessNextSection := ADR(chipboardSection);
	chipboardSection.accessNextSection := ADR(woodBunkSection);
	woodBunkSection.accessNextSection := ADR(outputSection);
	outputSection.accessNextSection := 0;
*)

initSections := TRUE;
END_METHOD

METHOD PRIVATE interpretTransmission : BOOL
VAR_INPUT
	data : REFERENCE TO AdsData;
END_VAR
VAR
	i : INT;
END_VAR
CASE data.description OF
	EventsEnum.BUNDLE_IN:
		MEMCPY(ADR(bundleIn), ADR(data.binaryData), SIZEOF(bundleIn));
			
	EventsEnum.BUNDLE_ETA:
		MEMCPY(ADR(expectedBundles[numEtaBundles]), ADR(data.binaryData), SIZEOF(expectedBundles[numEtaBundles]));
		expectedArrivals[numEtaBundles] := data.timestamp;
		
END_CASE
END_METHOD

METHOD maintenance : BOOL
VAR_INPUT
END_VAR
END_METHOD

METHOD PRIVATE process : BOOL
(*
full parallel processsing
all sections may operate concurrently on any bundle
*)
(*
paperSection(
	enable:= run[SectionEnum.PAPER], 
	bundlesQueue:= bundlesQueue, 
	bundlesBypass:= bundlesBypass,
	bundleOut=> , 
	bypass=> , 
	ready=> , 
	busy=> sectionsBusy[SectionEnum.PAPER], 
	done=> , 
	error=> , 
	backlog=> ,
	iBundle=> sectionsIterator[SectionEnum.PAPER],
	iPair=> );
	
cardboardCornerGuardSection(
	enable:= run[SectionEnum.CARDBOARD_CORNERGUARD],
	bundlesQueue:= bundlesQueue, 
	bundlesBypass:= bundlesBypass,
	bundleOut=> ,
	bypass=> , 
	ready=> , 
	busy=> sectionsBusy[SectionEnum.CARDBOARD_CORNERGUARD], 
	done=> , 
	error=> , 
	backlog=> ,
	iBundle=> sectionsIterator[SectionEnum.CARDBOARD_CORNERGUARD],
	iPair=> );

chipboardSection(
	enable:= run[SectionEnum.CHIPBOARD],
	bundlesQueue:= bundlesQueue, 
	bundlesBypass:= bundlesBypass, 
	bundleOut=> ,
	bypass=> , 
	ready=> , 
	busy=> sectionsBusy[SectionEnum.CHIPBOARD], 
	done=> , 
	error=> , 
	backlog=> ,
	iBundle=> sectionsIterator[SectionEnum.CHIPBOARD],
	iPair=> );
*)

(*
woodBunkSection(
	enable:= run[SectionEnum.WOOD_BUNK],
	bundlesQueue:= bundlesQueue, 
	bundlesBypass:= bundlesBypass, 
	bundleOut=> ,
	bypass=> , 
	ready=> , 
	busy=> sectionsBusy[SectionEnum.WOOD_BUNK], 
	done=> , 
	error=> , 
	backlog=> ,
	iBundle=> sectionsIterator[SectionEnum.WOOD_BUNK],
	iPair=> );
*)
(*
outputSection(
	enable:= run[SectionEnum.OUTPUT],
	bundlesQueue:= bundlesQueue, 
	bundlesBypass:= bundlesBypass,
	outputBuffer:= outputBuffer,
	bundleOut=> , 
	bypass=> , 
	ready=> , 
	busy=> sectionsBusy[SectionEnum.OUTPUT],
	done=> , 
	error=> , 
	backlog=> ,
	iBundle=> sectionsIterator[SectionEnum.OUTPUT],
	iPair=> );
*)
END_METHOD

METHOD PRIVATE ps_AbortCondition : BOOL
VAR_INPUT
END_VAR
END_METHOD

METHOD PRIVATE ps_Aborted : BOOL
VAR_INPUT
END_VAR
END_METHOD

METHOD PRIVATE ps_Aborting : BOOL
VAR_INPUT
END_VAR
END_METHOD

METHOD PRIVATE ps_Clearing : BOOL
VAR_INPUT
END_VAR
END_METHOD

METHOD PRIVATE ps_Complete : BOOL
VAR_INPUT
END_VAR
END_METHOD

METHOD PRIVATE ps_Completing : BOOL
VAR_INPUT
END_VAR
END_METHOD

METHOD PRIVATE ps_Execute : BOOL
VAR_INPUT
END_VAR
VAR_OUTPUT
	error : BOOL;
END_VAR
CASE pmlMode OF
	0: //invalid mode
	ePMLCustomUnitMode_Production:		ps_Execute := process();
	ePMLCustomUnitMode_Maintenance:		maintenance();
	ePMLCustomUnitMode_Manual:			//
	ePMLCustomUnitMode_SemiAuto:		ps_Execute := process(); //manually step bundle into area - sections may be auto while area is semi-auto
END_CASE
END_METHOD

METHOD PRIVATE ps_Held : BOOL
VAR_INPUT
END_VAR
END_METHOD

METHOD PRIVATE ps_HoldCondition : BOOL
VAR_INPUT
END_VAR
END_METHOD

METHOD PRIVATE ps_Holding : BOOL
VAR_INPUT
END_VAR
END_METHOD

METHOD PRIVATE ps_Idle : BOOL
VAR_INPUT
END_VAR
(*
IF BundleIsValid(currentBundle) THEN
	ps_Idle := TRUE;
	done := FALSE;
END_IF
*)

ps_Idle := TRUE; (*start section input*)
END_METHOD

METHOD PRIVATE ps_Resetting : BOOL
VAR_INPUT
END_VAR
END_METHOD

METHOD PRIVATE ps_Starting : BOOL
VAR_INPUT
END_VAR
END_METHOD

METHOD PRIVATE ps_StopCondition : BOOL
VAR_INPUT
END_VAR
END_METHOD

METHOD PRIVATE ps_Stopped : BOOL
VAR_INPUT
END_VAR
END_METHOD

METHOD PRIVATE ps_Stopping : BOOL
VAR_INPUT
END_VAR
END_METHOD

METHOD PRIVATE ps_SuspendCondition : BOOL
VAR_INPUT
END_VAR
END_METHOD

METHOD PRIVATE ps_Suspended : BOOL
VAR_INPUT
END_VAR
END_METHOD

METHOD PRIVATE ps_Suspending : BOOL
VAR_INPUT
END_VAR
END_METHOD

METHOD PRIVATE ps_Unholding : BOOL
VAR_INPUT
END_VAR
END_METHOD

METHOD PRIVATE ps_Unsuspending : BOOL
VAR_INPUT
END_VAR
END_METHOD

{attribute 'TcRpcEnable'}
METHOD PRIVATE receive : BOOL
VAR
	i : INT;
	shiftIndex : INT := -1;
	invalidBundle : Bundle;
END_VAR
FOR i:=0 TO CONSTS.maxQueue BY 1 DO //find the bundle in the ETA queue
	IF expectedBundles[i] = bundleIn.id THEN
		shiftIndex := i;
		EXIT;
	END_IF
END_FOR

IF shiftIndex > -1 THEN //if the bundle is found in the ETA queue, shift everything down
	MEMMOVE(
		ADR(expectedBundles[shiftIndex]), 
		ADR(expectedBundles[shiftIndex + 1]), 
		SIZEOF(STRING) * TO_UINT(CONSTS.maxQueue - shiftIndex));
		
	MEMMOVE(
		ADR(expectedArrivals[shiftIndex]), 
		ADR(expectedArrivals[shiftIndex + 1]), 
		SIZEOF(TIMESTRUCT) * TO_UINT(CONSTS.maxQueue - shiftIndex) );
		
	numEtaBundles := numEtaBundles - 1;
END_IF

FOR i:=0 TO CONSTS.maxQueue BY 1 DO
	IF BundleIsValid(bundlesQueue[i]) AND NOT bundlesBypass[i] THEN
		bundlesQueue[i] := bundleIn;
		bundlesBypass[i] := FALSE;
		
		receive := TRUE;
		RETURN;
	END_IF
END_FOR

IF NOT receive THEN
	error := TRUE;
END_IF
END_METHOD

METHOD PRIVATE runPML : BOOL
(*
PackML
	state machine for packaging applications - see Tc3_PackML_V2 library on InfoSys
	
	final states - wait for an input or condition and command to new state
	intermediate states - complete a task and call pmlStateMachine.M_StateComplete() to advance to next state
	
the following states currently use the same logic (albeit in different methods), implementation may change later
	ps_Stopping() and ps_Aborting()
	ps_Resetting() and ps_Clearing()
	
STOP - controlled stop **with intent to shutdown or vacate for extended time** induced by operator/HMI - otherwise use HOLD
ABORT - emergency stop due to machine errors


HOLD - minor local issues
SUSPEND - external issues

EXECUTE - major control logic
	different modes may require different tasks
	create methods as required for different modes, then call the correct method in ps_Completing()
	can be commanded to STOP, ABORT, HOLD, or SUSPEND at any point
COMPLETING - process complete, move product out of system and finish transition to COMPLETED

the implementation below can be copied to all POUs that use a PackML state machine
the individual ps_< > methods need to be implemented for the specific application
*)
IF ps_AbortCondition() THEN //abort condition
	pmlCommand := ePMLCommand_Abort;
ELSIF ps_StopCondition() THEN //stop condition
	pmlCommand := ePMLCommand_Stop;
END_IF

CASE pmlState OF
	0 (*ePMLState_Undefined*): //default state on startup
		pmlCommand := ePMLCommand_Stop;
		
	ePMLState_Stopping:
		IF ps_Stopping() THEN
			pmlStateMachine.M_StateComplete();
		END_IF
		
	ePMLState_Stopped:
		IF ps_Stopped() THEN
			pmlCommand := ePMLCommand_Reset;
		END_IF
	
    ePMLState_Resetting:
		IF ps_Resetting() THEN
			pmlStateMachine.M_StateComplete();
		END_IF
		
	ePMLState_Idle:
		IF ps_Idle() THEN
			pmlCommand := ePMLCommand_Start;
		END_IF		
	
	ePMLState_Starting:
		IF ps_Starting() THEN
			pmlStateMachine.M_StateComplete();
		END_IF
	
	ePMLState_Execute: //check the conditions in order of their priority, currently HOLD has the highest priority
		IF ps_HoldCondition() THEN
			pmlCommand := ePMLCommand_Hold;
			
		ELSIF ps_SuspendCondition() THEN
			pmlCommand := ePMLCommand_Suspend;			
		
		ELSIF ps_Execute(error => error) THEN //ps_Execute.error => THIS^.error
			pmlStateMachine.M_StateComplete();
			pmlCommand := ePMLCommand_Complete;
		END_IF
		
	ePMLState_Completing:
		IF ps_Completing() THEN
			pmlStateMachine.M_StateComplete();
		END_IF
	
	ePMLState_Complete:
		IF ps_Complete() THEN
			pmlCommand := ePMLCommand_Reset;
		END_IF
	
	ePMLState_Holding:
		IF ps_Holding() THEN
			pmlStateMachine.M_StateComplete();
		END_IF
	
	ePMLState_Held:
		IF NOT hold THEN
			pmlCommand := ePMLCommand_Unhold;
		END_IF
	
	ePMLState_Unholding:
		IF ps_Unholding() THEN
			pmlStateMachine.M_StateComplete(); //release all pause commands and IO
		END_IF
		
	ePMLState_Suspending: //based on next section conditions
		IF ps_Suspending() THEN
			pmlStateMachine.M_StateComplete();
		END_IF
		
	ePMLState_Suspended: //based on next section conditions
		IF ps_Suspended() THEN
			pmlCommand := ePMLCommand_Unsuspend;
		END_IF
	
	ePMLState_Unsuspending: //based on next section conditions
		IF ps_Unsuspending() THEN
			pmlStateMachine.M_StateComplete();
		END_IF
	
	ePMLState_Aborting:
		IF ps_Aborting() THEN
			pmlStateMachine.M_StateComplete();
		END_IF
	
	ePMLState_Aborted:
		IF ps_Aborted() THEN
			pmlCommand := ePMLCommand_Clear;
		END_IF
	
	ePMLState_Clearing:
		IF ps_Clearing() THEN
			pmlStateMachine.M_StateComplete();
		END_IF
	
END_CASE
END_METHOD

METHOD shiftBundles : BOOL
VAR_INPUT
END_VAR
//shift down parallel arrays
MEMMOVE(ADR(bundlesQueue[0]), ADR(bundlesQueue[1]), SIZEOF(Bundle) * TO_UINT(CONSTS.maxQueue));
MEMMOVE(ADR(bundlesBypass[0]), ADR(bundlesBypass[1]), SIZEOF(BOOL) * TO_UINT(CONSTS.maxQueue));

//decrement each section's iterator to realign with their correct bundle
//paperSection.shiftIterator();
//cardboardCornerGuardSection.shiftIterator();
//chipboardSection.shiftIterator();
woodBunkSection.shiftIterator();
//outputSection.shiftIterator();
END_METHOD

METHOD PRIVATE transfer : BOOL
VAR
	i : INT;
END_VAR
//send TCP/ADS transmission back to Dispatch once bundle is removed from the plant

IF clearPassBuffer THEN
	dbLogger.queueEvent(event:= EventsEnum.BUNDLE_OUT); //modify to include bundle ID
	//outputBufferPass := GVL.nullBundle;
	MEMSET(ADR(outputBufferPass), 0, SIZEOF(outputBufferPass));
END_IF

IF clearFailBuffer THEN
	dbLogger.queueEvent(event:= EventsEnum.BUNDLE_OUT); //modify to include bundle ID
	//outputBufferFail := GVL.nullBundle;
	MEMSET(ADR(outputBufferFail), 0, SIZEOF(outputBufferFail));
END_IF
END_METHOD

END_PROGRAM

// ---- Sections/A26 - Spacer Recollection/SpacerRecollectionUnit.TcPOU
FUNCTION_BLOCK SpacerRecollectionUnit //EXTENDS SectionEx
VAR_IN_OUT
	robot : RobotA26; //placeholder, will need another robot definition for A26
	robotSlider : ServoNC;
END_VAR
VAR_INPUT
	spacerPresent_A24_LRC_C02 : BOOL; //these conveyoors move bundles from A2.7 to A2.4
	spacerPresent_A24_LRC_C04 : BOOL;
	spacerPresent_A24_LRC_C06 : BOOL;
	spacerPresent_A24_LRC_C08 : BOOL;
	spacerPresent_A24_LRC_C10 : BOOL;
	spacerPresent_A24_LRC_C12 : BOOL;
END_VAR
VAR_OUTPUT
	ready : BOOL;
	busy : BOOL;
	done : BOOL;
	error : BOOL;
	
	failCounter : INT;
END_VAR
VAR
	//spacersPresent : ARRAY[1..6] OF BOOL;
	
	step : (IDLE, SLIDE, PICK_SPACER, COMPLETE);
	iPosition : INT;
END_VAR
VAR
	pos1, pos2, pos3 : LREAL;
END_VAR

ready := step = 0;
busy := step > 0;
done := done;
error := error;
(*
spacersPresent[1] := spacerPresent_A24_LRC_C02;
spacersPresent[2] := spacerPresent_A24_LRC_C04;
spacersPresent[3] := spacerPresent_A24_LRC_C06;
spacersPresent[4] := spacerPresent_A24_LRC_C08;
spacersPresent[5] := spacerPresent_A24_LRC_C10;
spacersPresent[6] := spacerPresent_A24_LRC_C12;
*)
IF 
	A24.A24_SC_C01.IsOccupied OR
	A24.A24_SC_C03.IsOccupied OR
	A24.A24_SC_C05.IsOccupied OR
	A24.A24_SC_C07.IsOccupied OR
	A24.A24_SC_C09.IsOccupied OR
	A24.A24_SC_C11.IsOccupied OR
	A24.A24_SC_C13.IsOccupied
THEN
	robot.clearCommand();
	
ELSE
	//remove spacers from transfer conveyors in ascending order
	process();
	
END_IF

METHOD process : BOOL
VAR_INPUT
END_VAR
VAR
	spacersPresent : ARRAY[1..6] OF BOOL := [
		spacerPresent_A24_LRC_C02,
		spacerPresent_A24_LRC_C04,
		spacerPresent_A24_LRC_C06,
		spacerPresent_A24_LRC_C08,
		spacerPresent_A24_LRC_C10,
		spacerPresent_A24_LRC_C12];
END_VAR
VAR CONSTANT
	suctionDistance : INT := 10;
END_VAR
{warning disable C0371}

iPosition := MAX(1, iPosition); //value is always at least 1

CASE step OF
	IDLE:
		IF DataIsEmpty(arr := ADR(spacersPresent), arrSize := SIZEOF(spacersPresent)) THEN
			iPosition := 0;
			failCounter := 0;
			process := TRUE;
		
		ELSIF NOT spacersPresent[iPosition] THEN
			iPosition := iPosition + 1;
			
		ELSIF robot.Ready THEN
			step := PICK_SPACER;
		END_IF
		
	PICK_SPACER:
		IF robot.eoatDistance > suctionDistance THEN
			robot.HoldMaterial := 'SPACER';
		ELSE
			robot.HoldMaterial := '';
		END_IF
	
		IF robot.Done THEN
			step := COMPLETE;
		ELSE
			robot.setGroup(group := 1, value := TaskA26.PICK_SPACER);
			robot.setGroup(group := 2, value := iPosition);
		END_IF
		
	COMPLETE:
		robot.HoldMaterial := '';
		
		IF spacersPresent[iPosition] THEN
			failCounter := failCounter + 1;
		END_IF
		
		robot.clearCommand();
		step := 0;
	
END_CASE
END_METHOD

END_FUNCTION_BLOCK

// ---- HARDWARE_DISTRUBUTION/A24.TcPOU
PROGRAM A24
VAR_OUTPUT //conveyors only
	A24_LRC_C02 	: Conveyor; //these conveyoors move bundles from A2.7 to A2.4
	A24_LRC_C04 	: Conveyor;
	A24_LRC_C06	 	: Conveyor;
	A24_LRC_C08 	: Conveyor;
	A24_LRC_C10 	: Conveyor;
	A24_LRC_C12 	: Conveyor;
	
	A24_SC_C01 		: ConveyorSC; //these conveyors move bundles on A2.4 forward down the cell
	A24_SC_C03 		: ConveyorSC;
	A24_SC_C05 		: ConveyorSC;
	A24_SC_C07 		: ConveyorSC;
	A24_SC_C09 		: ConveyorSC;
	A24_SC_C11 		: ConveyorSC;
	A24_SC_C13 		: ConveyorSC;
END_VAR

END_PROGRAM

// ---- Sections/A22 - Cardboard/CardboardEx.TcPOU
FUNCTION_BLOCK CardboardEx EXTENDS SectionEx
VAR_IN_OUT
	benderLeft : FoldingMachine;
	
	robotLeft, robotRight : RobotA22;
	
	skidLeft, skidRight : SkidMagazine;
	magazineLeft, magazineRight : SkidMagazine;
	
	wrapper : WrapMachine;
	
	insertionLeft, insertionRight : Insertion;
	pistonBottom : SimplePiston;
	
	suctionTopLeft : ARRAY[*] OF SuctionPad; (*1..3*)
	suctionTopRight : ARRAY[*] OF SuctionPad; (*1..3*)
	suctionBottomLeft : ARRAY[*] OF SuctionPad; (*1..3*)
	suctionBottomRight : ARRAY[*] OF SuctionPad; (*1..3*)
	
	suctionBottom : ARRAY[*] OF SuctionPad; (*1..2*)
END_VAR
VAR	
	step : (IDLE, LOAD_SIDES_CORNERS, LOAD_TOP_BOTTOM, PUSH, TARGET_WRAP_POSITION, WRAP_AND_RELEASE, COMPLETE := 1050);
	
	masterLoadStep : INT;
	loadStepLeft, loadStepRight : INT;
	
	iWrap : INT;
	wrapPoints : INT;
	wrapRotations : INT;
	masterLength : INT;
	
	releaseDelayTimer : TON;
END_VAR
VAR //local types
	topLeftFoldsArr, topRightFoldsArr, bottomLeftFoldsArr, bottomRightFoldsArr : ARRAY[0..CONSTS.maxPairs] OF INT;
	
	//materialsArr : ARRAY[0..Consts.maxPairs] OF PositionMaterials;
	materialsArr : ARRAY[0..2*Consts.maxPairs] OF PositionMaterials;
	
	recipesCombined : BOOL;
	
	demoHeight : REAL := 640; //mm
	
	innerLoadedMaterials, outerLoadedMaterials : ARRAY[Surface.TOP..Surface.BOTTOM_RIGHT] OF STRING;
	//inner: cardboard by default
	//outer: corner guard by default
END_VAR
VAR CONSTANT
	releaseDelay : TIME := T#2000MS;
END_VAR
VAR
	//AOIs encapsulate functionality and reduce the number of module variables
	aoiCornerGuardLeft, aoiCornerGuardRight : AOI_LoadCornerGuard;
	aoiCornerCardboardLeft, aoiCornerCardboardRight : AOI_LoadCornerCardboard;
	aoiFlatCardboardLeft, aoiFlatCardboardRight : AOI_LoadFlatCardboard;
	
	//for testing only
	latchLeft, latchRight : BOOL; //prevents sliders from overshooting the inner limit sensor
	suctionEnableTopLeft, suctionEnableTopRight, suctionEnableBottomLeft, suctionEnableBottomRight : BOOL;
END_VAR

aoiBlocks();

SUPER^();

METHOD PROTECTED aoiBlocks : BOOL
VAR_INPUT
END_VAR
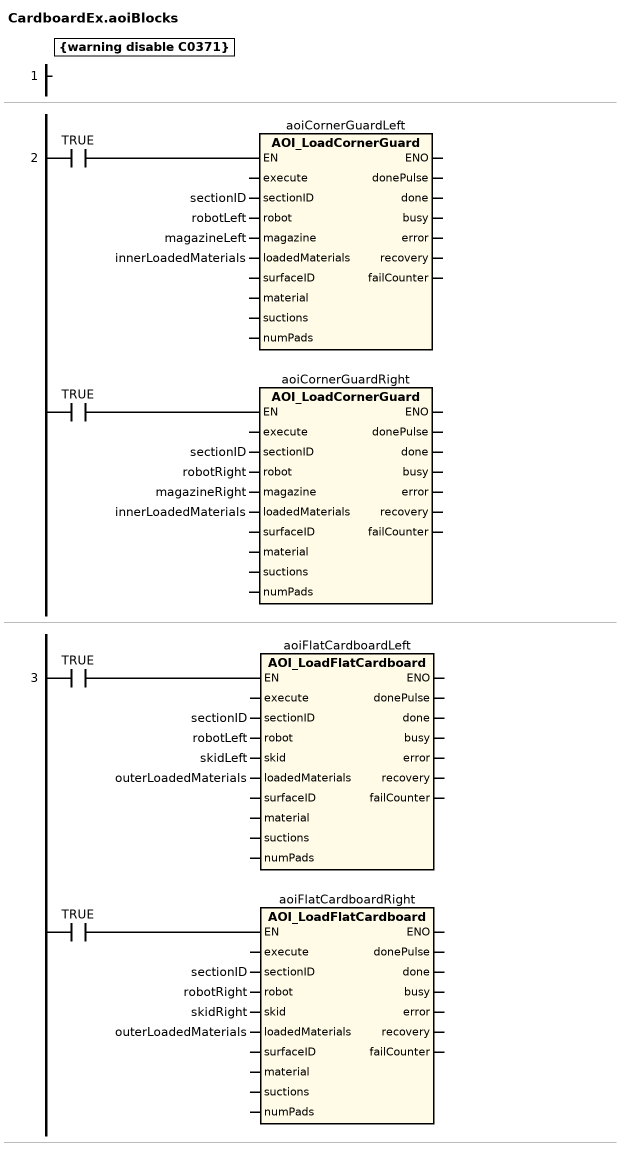
// NETWORK 1
// label: {warning disable C0371}

// NETWORK 2
aoiCornerGuardLeft(
    sectionID := sectionID,
    robot := robotLeft,
    magazine := magazineLeft,
    loadedMaterials := innerLoadedMaterials); // AOI_LoadCornerGuard
aoiCornerGuardRight(
    sectionID := sectionID,
    robot := robotRight,
    magazine := magazineRight,
    loadedMaterials := innerLoadedMaterials); // AOI_LoadCornerGuard

// NETWORK 3
aoiFlatCardboardLeft(
    sectionID := sectionID,
    robot := robotLeft,
    skid := skidLeft,
    loadedMaterials := outerLoadedMaterials); // AOI_LoadFlatCardboard
aoiFlatCardboardRight(
    sectionID := sectionID,
    robot := robotRight,
    skid := skidRight,
    loadedMaterials := outerLoadedMaterials); // AOI_LoadFlatCardboard
END_METHOD

METHOD PROTECTED combine : BOOL
VAR_IN_OUT
	cardboard : ARRAY[*] OF PositionMaterials;
	cornerGuard : ARRAY[*] OF PositionMaterials;
	
	combined : ARRAY[*] OF PositionMaterials;
END_VAR
VAR_INPUT
	cardboard_over_cornerGuard : BOOL;
END_VAR
VAR_INST
	topLength : REAL;
	leftLength : REAL;
	rightLength : REAL;
	bottomLength : REAL;
	
	topLeftLength : REAL;
	topRightLength : REAL;
	bottomLeftLength : REAL;
	bottomRightLength : REAL;
	
	outerMaterialLength : REAL;
	innerMaterialLength : REAL;
	
	i : INT;
	iCardboard : INT;
	iCornerGuard : INT;
END_VAR
FOR i:=0 TO CONSTS.maxPairs*2 BY 1 DO
	IF //no more cardboard (reached end of array or unused entries), 
		(iCardboard >= CONSTS.maxPairs OR_ELSE NOT PositionIsValid(cardboard[iCardboard])) AND_THEN //no more valid cardboard entries
		iCornerGuard < CONSTS.maxPairs AND_THEN //still has remaining corner guard
		PositionIsValid(cornerGuard[iCornerGuard]) //remaining corner guard is valid		
	THEN //finish with cornerguard
		combined[i] := cornerGuard[iCornerGuard];
		iCornerGuard := iCornerGuard + 1;
		CONTINUE;
	END_IF
	
	IF //no more cornerguard (reached end of array or unused entries)
		(iCornerGuard >= CONSTS.maxPairs OR_ELSE NOT PositionIsValid(cornerGuard[iCornerGuard])) AND_THEN
		iCardboard < CONSTS.maxPairs AND_THEN
		PositionIsValid(cardboard[iCardboard])
	THEN //finish with cardboard
		combined[i] := cardboard[iCardboard];
		iCardboard := iCardboard + 1;
		CONTINUE;
	END_IF
	
	(*
	IF NOT cardboard_over_cornerGuard THEN //cardboard on inside
		setOrder(cardboard, cornerGuard, combined, iCardboard, iCornerGuard, i);
		
	ELSE //cardboard on outside
		setOrder(cornerGuard, cardboard, combined, iCornerGuard, iCardboard, i);
		
	END_IF
	*)
END_FOR

combine := TRUE;
END_METHOD

METHOD PROTECTED load : BOOL
VAR_INPUT
	pairIndex : INT;
END_VAR
VAR_OUTPUT
	error : BOOL;
END_VAR
VAR
	pair : REFERENCE TO PositionMaterials REF= materialsArr[pairIndex];
	nextPair : REFERENCE TO PositionMaterials;
END_VAR
(*
unlike other sections, the load() function for cardboard + corner guard only loads the corners
to load flat cardboards, use the function loadFlats()
*)
{warning disable C0371}

IF robotLeft.error OR robotRight.error THEN
	RETURN;
ELSIF NOT (robotLeft.reserve(sectionID) AND robotRight.reserve(sectionID)) THEN //both robots must be reserved first
	RETURN;
END_IF

IF pairIndex + 1 < CONSTS.maxPairs THEN
	nextPair REF= materialsArr[pairIndex + 1];
END_IF

CASE masterLoadStep OF
	0: //load this pair's side cardboards
		masterLoadStep := 10;
		IF
			loadFlatCardboardsEx(
				robot:= robotLeft, 
				aoiLoad:= aoiFlatCardboardLeft, 
				loadStep:= loadStepLeft, 
				pairIndex:= pairIndex, 
				includeTop:= FALSE, 
				includeLeft:= TRUE, 
				includeRight:= FALSE, 
				includeBottom:= FALSE, 
				error=> )
			AND
			loadFlatCardboardsEx(
				robot:= robotLeft, 
				aoiLoad:= aoiFlatCardboardLeft, 
				loadStep:= loadStepLeft, 
				pairIndex:= pairIndex, 
				includeTop:= FALSE, 
				includeLeft:= FALSE, 
				includeRight:= TRUE, 
				includeBottom:= FALSE, 
				error=> )
		THEN
			masterLoadStep := 10;
			loadStepLeft := loadStepRight := 0;
		END_IF
		
		
	10: //next pair (which is to be placed over this pair) has the same position as this pair
		IF pairIndex + 1 >= CONSTS.maxPairs THEN //no next pair - final pair is index 15 (16-1), not 16
			masterLoadStep := 20;
			loadStepLeft := loadStepRight := 0;
			
		ELSIF pair.position < nextPair.position THEN
			masterLoadStep := 20;
			loadStepLeft := loadStepRight := 0;
		(*	
		ELSIF MatchesMaterialType(pair:= nextPair, materialType:= 'CAR') AND_THEN loadCornerCardboards(pairIndex:= pairIndex + 1) THEN
			masterLoadStep := 20;
			loadStepLeft := loadStepRight := 0;
		*)
		ELSIF MatchesMaterialType(pair:= nextPair, materialType:= 'COR') AND_THEN loadCornerGuards(pairIndex:= pairIndex + 1) THEN
			masterLoadStep := 20;
			loadStepLeft := loadStepRight := 0;
			
		END_IF
		
	20: //load current pair
		IF
			MatchesMaterialType(pair:= pair, materialType:= 'CAR') AND_THEN loadCornerCardboards(pairIndex:= iPair) OR_ELSE
			MatchesMaterialType(pair:= pair, materialType:= 'COR') AND_THEN loadCornerGuards(pairIndex:= iPair)
		THEN //is cardboard
			loadStepLeft := loadStepRight := 0;
			masterLoadStep := COMPLETE;
		END_IF
	
	COMPLETE:
		robotLeft.release(sectionID);
		robotRight.release(sectionID);
		
		loadStepLeft := loadStepRight := 0;
		masterLoadStep := 0;
		load := TRUE;
	
END_CASE
END_METHOD

METHOD PROTECTED loadCornerCardboards : BOOL
VAR_INPUT
	pairIndex : INT;
END_VAR
VAR_OUTPUT
	error : BOOL;
END_VAR
VAR
	errorLeft, errorRight : BOOL;
	leftSuctionArr, rightSuctionArr : POINTER TO SuctionPad;
	leftNextSet, rightNextSet : INT;
	leftMaterial, rightMaterial : STRING;
	leftFold, rightFold : INT;
	
	pair : REFERENCE TO PositionMaterials REF= materialsArr[pairIndex];
	topLeftFold : INT := topLeftFoldsArr[pairIndex];
	topRightFold : INT := topRightFoldsArr[pairIndex];
	bottomLeftFold : INT := bottomLeftFoldsArr[pairIndex];
	bottomRightFold : INT := bottomRightFoldsArr[pairIndex];
END_VAR
{warning disable C0371}

loadCornerCardboards := 
	loadCornerCardboardsEx(
		robot:= robotLeft, 
		aoiLoad:= aoiCornerCardboardLeft, 
		loadStep:= loadStepLeft, 
		pairIndex:= pairIndex, 
		includeTopLeft:= TRUE, 
		includeTopRight:= FALSE, 
		includeBottomLeft:= TRUE, 
		includeBottomRight:= FALSE, 
		error=> errorLeft)
	AND
	loadCornerCardboardsEx(
		robot:= robotRight, 
		aoiLoad:= aoiCornerCardboardRight, 
		loadStep:= loadStepRight, 
		pairIndex:= pairIndex, 
		includeTopLeft:= FALSE, 
		includeTopRight:= TRUE, 
		includeBottomLeft:= FALSE, 
		includeBottomRight:= TRUE, 
		error=> errorLeft);
		
error := errorLeft OR errorRight;

(*
CASE cornerSetLeft OF
	0:
		leftNextSet := Surface.TOP_RIGHT;
		cornerSetLeft := 0;
		
	Surface.TOP_RIGHT: 
		leftNextSet := Surface.TOP_LEFT;
		leftSuctionArr := suctionTopRight;
		leftMaterial := pair.topRight;
		leftFold := topRightFold;
		
	Surface.TOP_LEFT: 
		leftNextSet := Surface.BOTTOM_RIGHT;
		leftSuctionArr := suctionTopLeft;
		leftMaterial := pair.topLeft;
		leftFold := topLeftFold;
		
	Surface.BOTTOM_RIGHT:
		leftNextSet := Surface.BOTTOM_LEFT;
		leftSuctionArr := suctionBottomRight;
		leftMaterial := pair.bottomRight;
		leftFold := bottomRightFold;
		
	Surface.BOTTOM_LEFT: 
		leftNextSet := COMPLETE;
		leftSuctionArr := suctionBottomLeft;
		leftMaterial := pair.bottomLeft;
		leftFold := bottomLeftFold;
END_CASE
IF
	(cornerSetLeft = 0 OR cornerSetLeft = COMPLETE) OR_ELSE
	leftCornerSequence(
		robot:= robotLeft, 
		skid:= skidLeft, 
		suctions := leftSuctionArr,
		loadStep:= loadStepLeft, 
		surfaceID:= cornerSetLeft,
		material:= pair.topRight, 
		foldPos0:= topRightFold, 
		foldPos1:= 0, 
		error=> )
THEN
	cornerSetLeft := leftNextSet;
	loadStepLeft := 0;
END_IF


CASE cornerSetRight OF
	0:
		cornerSetRight := Surface.TOP_RIGHT;
		rightSuctionArr := suctionTopRight;
		
	Surface.TOP_RIGHT:		
		rightNextSet := Surface.BOTTOM_RIGHT;
		rightSuctionArr := suctionTopRight;
		rightMaterial := pair.topRight;
		rightFold := topRightFold;
		
	Surface.BOTTOM_RIGHT: 
		rightNextSet := COMPLETE;
		rightSuctionArr := suctionBottomRight;
		rightMaterial := pair.bottomRight;
		rightFold := bottomRightFold;		
END_CASE
IF
	(cornerSetRight = 0 OR cornerSetRight = COMPLETE) OR_ELSE
	rightCornerSequence(
		robot:= robotRight, 
		skid:= skidRight, 
		suctions := rightSuctionArr,
		loadStep:= loadStepRight, 
		material:= pair.topRight, 
		surfaceID:= cornerSetRight,
		foldPos0:= pair.topRightFold, 
		foldPos1:= 0, 
		error=> )
THEN
	cornerSetRight := rightNextSet;
	loadStepRight := 0;
END_IF



IF cornerSetLeft = COMPLETE AND cornerSetRight = COMPLETE THEN
	loadCornerCardboards := TRUE;
	
	loadStepLeft := loadStepRight := 0;
	cornerSetLeft := cornerSetRight := 0;
END_IF
*)
END_METHOD

METHOD PROTECTED loadCornerCardboardsEx : BOOL
VAR_IN_OUT
	robot : RobotA22;
	aoiLoad : AOI_LoadCornerCardboard;
	loadStep : INT;
END_VAR
VAR_INPUT
	pairIndex : INT;
	includeTopLeft, includeTopRight, includeBottomLeft, includeBottomRight : BOOL;
END_VAR
VAR_OUTPUT
	error : BOOL;
END_VAR
VAR
	suctionsArrLeft, suctionsArrRight : POINTER TO SuctionPad;
	nextSetLeft, nextSetRight : INT;

	pair : REFERENCE TO PositionMaterials REF= materialsArr[pairIndex];
	topLeftFold : INT := topLeftFoldsArr[pairIndex];
	topRightFold : INT := topRightFoldsArr[pairIndex];
	bottomLeftFold : INT := bottomLeftFoldsArr[pairIndex];
	bottomRightFold : INT := bottomRightFoldsArr[pairIndex];
END_VAR
{warning disable C0371}

IF robot.error THEN
	error := TRUE;
	RETURN;
ELSIF robot.reservation <> sectionID AND_THEN NOT robot.reserve(sectionID) THEN
	RETURN;
ELSIF robot.tool <> sectionID AND_THEN NOT robot.changeEOAT(targetTool := sectionID) THEN
	RETURN;
END_IF

error := aoiLoad.error;

CASE loadStep OF
	0:
		loadStep := Surface.BOTTOM_LEFT;
		
	Surface.BOTTOM_LEFT:
		IF NOT includeBottomLeft OR aoiLoad.donePulse THEN
			aoiLoad.execute := FALSE;
			aoiLoad.material := '';
			loadStep := Surface.BOTTOM_RIGHT;
			RETURN;
		END_IF
		
		aoiLoad.surfaceID := loadStep;
		aoiLoad.material := pair.bottomLeft;
		aoiLoad.suctions := suctionBottomLeft;
		aoiLoad.numPads := UPPER_BOUND(suctionBottomLeft, 1) - LOWER_BOUND(suctionBottomLeft, 1) + 1;
		
		aoiLoad.foldPos0 := bottomLeftFold;
		aoiLoad.foldPos1 := 0;
		
		aoiLoad.execute := NOT aoiLoad.busy;
		
	Surface.BOTTOM_RIGHT:
		IF NOT includeBottomRight OR aoiLoad.donePulse THEN
			aoiLoad.execute := FALSE;
			aoiLoad.material := '';
			loadStep := Surface.TOP_LEFT;
			RETURN;
		END_IF
		
		aoiLoad.surfaceID := loadStep;
		aoiLoad.material := pair.bottomRight;
		aoiLoad.suctions := suctionBottomRight;
		aoiLoad.numPads := UPPER_BOUND(suctionBottomRight, 1) - LOWER_BOUND(suctionBottomRight, 1) + 1;
		
		aoiLoad.foldPos0 := bottomRightFold;
		aoiLoad.foldPos1 := 0;
		
		aoiLoad.execute := NOT aoiLoad.busy;
	
	Surface.TOP_LEFT:		
		IF NOT includeTopLeft OR aoiLoad.donePulse THEN
			aoiLoad.execute := FALSE;
			aoiLoad.material := '';
			loadStep := Surface.TOP_RIGHT;
			RETURN;
		END_IF
		
		aoiLoad.surfaceID := loadStep;
		aoiLoad.material := pair.top;
		aoiLoad.suctions := suctionTopLeft;
		aoiLoad.numPads := UPPER_BOUND(suctionTopLeft, 1) - LOWER_BOUND(suctionTopLeft, 1) + 1;
		
		aoiLoad.foldPos0 := topLeftFold;
		aoiLoad.foldPos1 := 0;
		
		aoiLoad.execute := NOT aoiLoad.busy;
		
	Surface.TOP_RIGHT:
		IF NOT includeTopRight OR aoiLoad.donePulse THEN
			aoiLoad.execute := FALSE;
			aoiLoad.material := '';
			loadStep := COMPLETE;
			RETURN;
		END_IF
		
		aoiLoad.surfaceID := loadStep;
		aoiLoad.material := pair.topRight;
		aoiLoad.suctions := suctionTopRight;
		aoiLoad.numPads := UPPER_BOUND(suctionTopRight, 1) - LOWER_BOUND(suctionTopRight, 1) + 1;
		
		aoiLoad.foldPos0 := topRightFold;
		aoiLoad.foldPos1 := 0;
		
		aoiLoad.execute := NOT aoiLoad.busy;
		
